Yaskawa INFORM job: SKRZYNIA_5040_90_STOPNI_10BR_OLD.JBI

/JOB
//NAME SKRZYNIA_5040_90_STOPNI_10BR_OLD
//POS
///NPOS 659,659,0,49,0,0
///TOOL 0
///POSTYPE PULSE
///PULSE
C00000=0,-52280,40443,0,6876,0
C00001=82314,-24956,17040,59626,-27382,6248
C00002=93910,-8625,17040,59626,-43355,6248
C00003=98846,-1061,-42166,80308,-57081,-16120
C00004=100452,6057,-48127,85711,-56704,-21322
C00005=96349,29000,-36127,85072,-63022,-26262
C00006=95580,33075,-33256,84644,-64024,-26851
C00007=94197,33846,-32020,85210,-63413,-26698
C00008=95580,33075,-33256,84644,-64024,-26851
C00009=94888,31114,-36362,85298,-63687,-27185
C00010=95580,33075,-33256,84644,-64024,-26851
C00011=95263,33142,-33256,84677,-63995,-26850
C00012=94634,33491,-32695,84935,-63717,-26781
C00013=94130,33776,-32235,85140,-63494,-26725
C00014=95104,32689,-33981,84829,-63917,-26928
C00015=94679,31503,-35865,85229,-63711,-27129
C00016=95263,33142,-33256,84677,-63995,-26850
C00017=95260,33144,-33256,84678,-63995,-26850
C00018=94650,33483,-32714,84929,-63727,-26783
C00019=94112,33789,-32223,85148,-63489,-26723
C00020=95084,32644,-34054,84845,-63909,-26937
C00021=94657,31449,-35950,85247,-63703,-27139
C00022=95260,33144,-33256,84678,-63995,-26850
C00023=95258,33145,-33257,84676,-63996,-26846
C00024=94953,33314,-32988,84801,-63862,-26812
C00025=94037,33833,-32158,85174,-63457,-26709
C00026=94978,32352,-34521,84941,-63860,-26983
C00027=94597,31295,-36193,85297,-63678,-27162
C00028=95258,33145,-33257,84676,-63996,-26846
C00029=95258,33145,-33257,84676,-63996,-26846
C00030=94635,33491,-32703,84932,-63720,-26777
C00031=94255,33706,-32357,85087,-63552,-26734
C00032=95076,32627,-34084,84849,-63906,-26937
C00033=94616,31344,-36119,85281,-63684,-27155
C00034=95258,33145,-33257,84676,-63996,-26846
C00035=95258,25631,32269,66559,-75499,-2416
C00036=95045,25799,32513,66531,-75379,-2372
C00037=94321,26382,33365,66429,-74973,-2219
C00038=95048,24784,31042,66584,-75290,-2483
C00039=94601,23046,28557,66633,-74859,-2609
C00040=95258,25631,32269,66559,-75499,-2416
C00041=98646,19496,-17631,99827,-80462,-21224
C00042=98317,21326,-15127,99395,-81089,-20992
C00043=97962,21529,-14845,99504,-80870,-20995
C00044=98567,20146,-16748,99341,-81286,-21080
C00045=98203,18829,-18537,99489,-81121,-21211
C00046=98811,21047,-15512,99242,-81394,-20987
C00047=98811,19937,1242,97498,-78933,-15296
C00048=98811,19937,1242,97498,-78933,-15296
C00049=98014,20416,1894,97635,-78400,-15298
C00050=98593,19084,88,97564,-78819,-15379
C00051=98194,17557,-1953,97683,-78607,-15521
C00052=98811,19937,1242,97498,-78933,-15296
C00053=98765,34858,63506,90961,-74847,-417
C00054=98962,39103,70654,91062,-76265,452
C00055=98093,40155,72476,90768,-75677,655
C00056=98962,39103,70654,91062,-76265,452
C00057=98539,36034,65455,91246,-76081,-158
C00058=98962,39103,70654,91062,-76265,452
C00059=98994,31803,58419,90917,-73461,-1055
C00060=94428,854,16076,89248,-50738,-4740
C00061=88080,-20128,-3199,80943,-31244,-2335
C00062=48287,-44591,-17414,16172,-14532,25809
C00063=48287,-44591,-17414,16172,-14532,25809
C00064=85348,-13130,13838,41209,-47455,8220
C00065=99199,18818,35660,68259,-73735,-6208
C00066=95720,15423,18785,70454,-68603,-10022
C00067=95720,15423,18785,70454,-68603,-10022
C00068=97055,28839,36684,71776,-79389,-10554
C00069=95990,29701,37981,71658,-78759,-10350
C00070=97055,28839,36684,71776,-79389,-10554
C00071=96570,26656,33448,71832,-78908,-10775
C00072=97055,28839,36684,71776,-79389,-10554
C00073=97055,28839,36684,71776,-79389,-10554
C00074=97055,28839,36684,71776,-79389,-10554
C00075=96028,29668,37934,71662,-78782,-10355
C00076=97055,28839,36684,71776,-79389,-10554
C00077=96569,26658,33449,71833,-78910,-10776
C00078=97055,28839,36684,71776,-79389,-10554
C00079=97055,28839,36684,71776,-79389,-10554
C00080=97055,28839,36684,71776,-79389,-10554
C00081=96073,29634,37879,71669,-78808,-10363
C00082=97055,28839,36684,71776,-79389,-10554
C00083=96556,26588,33346,71835,-78895,-10784
C00084=97055,28839,36684,71776,-79389,-10554
C00085=97055,28839,36684,71776,-79389,-10554
C00086=97055,28839,36684,71776,-79389,-10554
C00087=96070,29634,37881,71667,-78806,-10365
C00088=97055,28839,36684,71776,-79389,-10554
C00089=96542,26531,33264,71837,-78884,-10788
C00090=97055,28839,36684,71776,-79389,-10554
C00091=99222,23346,17795,82202,-78388,4176
C00092=99222,23346,17795,82202,-78388,4176
C00093=98198,24012,18735,82231,-77709,4276
C00094=99222,23346,17795,82202,-78388,4176
C00095=98846,21740,15549,82282,-78105,4028
C00096=99222,23346,17795,82202,-78388,4176
C00097=97305,19304,15511,100837,-75687,4760
C00098=97826,25373,24000,100195,-79238,5786
C00099=96887,26043,24967,100223,-78578,5793
C00100=97826,25373,24000,100195,-79238,5786
C00101=97448,23764,21701,100276,-79072,5588
C00102=97826,25373,24000,100195,-79238,5786
C00103=97826,25373,24000,100195,-79238,5786
C00104=97826,25373,24000,100195,-79238,5786
C00105=96843,26076,25015,100223,-78545,5791
C00106=97826,25373,24000,100195,-79238,5786
C00107=97441,23730,21652,100278,-79068,5583
C00108=97826,25373,24000,100195,-79238,5786
C00109=100071,8792,-2363,102947,-71408,2025
C00110=90699,-12620,-30080,113827,-52438,-6201
C00111=97832,-16290,-36993,112551,-57584,-6005
C00112=83036,-26396,-56580,138157,-49269,-16960
C00113=83036,-26453,-52828,136768,-47205,-15962
C00114=60067,-65836,-77869,147206,-28305,-20439
C00115=63330,-26972,24478,18707,-56801,31483
C00116=95462,-32664,-40336,69376,-39980,4046
C00117=100465,-3562,-10252,69901,-61773,-201
C00118=99635,18997,3540,80919,-74698,-6325
C00119=98097,22561,8426,80415,-76730,-6116
C00120=98097,22561,8426,80415,-76730,-6116
C00121=97377,23028,9077,80478,-76265,-6042
C00122=98097,22561,8426,80415,-76730,-6116
C00123=97807,21406,6827,80497,-76510,-6215
C00124=98097,22561,8426,80415,-76730,-6116
C00125=98899,30801,44624,87834,-79065,838
C00126=98899,30801,44624,87834,-79065,838
C00127=98247,31325,45433,87747,-78622,912
C00128=98899,30801,44624,87834,-79065,838
C00129=98602,29264,42279,87883,-78869,621
C00130=98899,30801,44624,87834,-79065,838
C00131=97973,11446,12587,89117,-68519,-2848
C00132=79911,-29338,-29911,88184,-26074,-2635
C00133=44299,-53382,-38573,-8929,-12050,42418
C00134=44299,-51091,-32799,-7549,-14278,41753
C00135=42754,-66126,12236,-1301,3231,7194
C00136=0,-52280,40443,0,6876,0
C00137=0,-52280,40443,0,6876,0
C00138=0,-43112,23163,-32261,-40956,-29092
C00139=48283,-21883,28214,25170,-26491,-48363
C00140=46664,-3144,58041,18842,-32105,-45325
C00141=50347,-18571,12268,49104,-16423,-60029
C00142=51149,-18702,10839,52647,-16284,-61663
C00143=49023,-16654,12458,50505,-14948,-60880
C00144=50458,-16314,12735,52976,-15639,-61913
C00145=50509,-19000,10610,51503,-15997,-61182
C00146=50509,-19000,10610,51503,-15997,-61182
C00147=51153,-18191,11234,52953,-16222,-61812
C00148=49506,-16603,12499,51322,-15186,-61219
C00149=50699,-16390,12671,53298,-15774,-62041
C00150=50704,-18403,11069,52157,-16018,-61478
C00151=50704,-18403,11069,52157,-16018,-61478
C00152=51011,-18259,11181,52703,-16157,-61707
C00153=49372,-16676,12437,51065,-15128,-61110
C00154=50855,-16321,12727,53567,-15849,-62152
C00155=50704,-18403,11069,52157,-16018,-61478
C00156=50704,-18403,11069,52157,-16018,-61478
C00157=51194,-17966,11787,52443,-16367,-61556
C00158=49641,-16469,12982,50879,-15396,-60984
C00159=51159,-16110,13274,53409,-16135,-62034
C00160=51194,-19029,8982,55593,-15729,-63095
C00161=51005,-17995,11387,52847,-16122,-61778
C00162=51030,-17982,11395,52891,-16135,-61798
C00163=49666,-16664,12446,51542,-15278,-61306
C00164=51234,-16283,12753,54139,-16047,-62382
C00165=51030,-17982,11395,52891,-16135,-61798
C00166=51030,-17982,11395,52891,-16135,-61798
C00167=51056,-17951,11420,52949,-16145,-61823
C00168=49507,-16445,12622,51407,-15172,-61259
C00169=51212,-15994,12989,54262,-16005,-62444
C00170=51056,-17951,11420,52949,-16145,-61823
C00171=50945,-18019,11363,52741,-16103,-61737
C00172=51451,-18380,9957,55416,-15976,-62984
C00173=49638,-16617,11364,53777,-14815,-62399
C00174=51249,-16205,11700,56405,-15635,-63491
C00175=50945,-18019,11363,52741,-16103,-61737
C00176=50945,-18019,11363,52741,-16103,-61737
C00177=51751,-18888,8325,57986,-15754,-64205
C00178=49901,-17096,9744,56519,-14545,-63700
C00179=51443,-16713,10055,58931,-15359,-64698
C00180=50945,-18019,11363,52741,-16103,-61737
C00181=50945,-18019,11363,52741,-16103,-61737
C00182=51752,-17629,11670,54137,-16475,-62321
C00183=49778,-15710,13222,52239,-15234,-61634
C00184=51536,-15216,13634,55124,-16102,-62830
C00185=50945,-18019,11363,52741,-16103,-61737
C00186=50028,-22953,-3957,22347,-31919,-54220
C00187=50556,-22259,-3444,23037,-31901,-54554
C00188=48685,-20311,-1961,21193,-31011,-53711
C00189=50316,-19877,-1623,23110,-31344,-54618
C00190=49456,-22793,-3840,21729,-31736,-53932
C00191=49763,-25421,-36239,24565,-26935,-60445
C00192=49763,-25421,-36239,24565,-26935,-60445
C00193=47682,-22631,-34091,22709,-25786,-59390
C00194=49411,-21994,-33587,24802,-26153,-60557
C00195=49763,-25421,-36239,24565,-26935,-60445
C00196=50713,-12366,-58367,41124,-17813,-74400
C00197=50531,-11018,-57111,41258,-17631,-74434
C00198=49339,-9106,-55286,40470,-17030,-73839
C00199=50327,-8799,-54988,41498,-17395,-74518
C00200=50078,-11370,-57441,40744,-17481,-74102
C00201=49763,-25421,-36239,24565,-26935,-60445
C00202=49426,-25689,-5908,21254,-32432,-53672
C00203=45389,-28224,4312,35967,-15579,-54278
C00204=40154,-51179,-915,24203,-8234,-36524
C00205=0,-52280,40443,0,6876,0
C00206=0,-52280,40443,0,6876,0
C00207=2117,-50103,-33543,4117,45077,-85249
C00208=-26439,-48928,-33543,4117,-52362,-85249
C00209=-26439,-27355,-33543,41485,-52362,-85249
C00210=-47486,-18593,-22655,32887,-41344,-78763
C00211=-48804,2873,-12100,24189,-42468,-81113
C00212=-46457,7101,-11330,26648,-40775,-82885
C00213=-47278,8641,-9483,26175,-40625,-82510
C00214=-46717,9819,-8044,26408,-40882,-82710
C00215=-47278,8641,-9483,26175,-40625,-82510
C00216=-48464,9694,-8203,25521,-40353,-81986
C00217=-47278,8641,-9483,26175,-40625,-82510
C00218=-44522,-635,-31983,49264,-28311,-89687
C00219=-44904,-149,-31453,49090,-28120,-89538
C00220=-44398,873,-30329,49324,-28371,-89731
C00221=-44904,-149,-31453,49090,-28120,-89538
C00222=-45751,485,-30759,48680,-27706,-89207
C00223=-44904,-149,-31453,49090,-28120,-89538
C00224=-41365,-13075,-22481,51159,-38446,-84131
C00225=-20796,-2039,-9686,94158,-57077,-89438
C00226=-24380,-971,-8542,94589,-54660,-89617
C00227=-25651,-542,-8077,94748,-53804,-89683
C00228=-25378,473,-6965,94714,-53986,-89667
C00229=-25651,-542,-8077,94748,-53804,-89683
C00230=-26467,-222,-7729,94854,-53254,-89725
C00231=-25651,-542,-8077,94748,-53804,-89683
C00232=-25651,-542,-8077,94748,-53804,-89683
C00233=-25946,-428,-7954,94785,-53605,-89698
C00234=-25690,517,-6922,94753,-53778,-89686
C00235=-25946,-428,-7954,94785,-53605,-89698
C00236=-26504,-206,-7715,94856,-53230,-89728
C00237=-25946,-428,-7954,94785,-53605,-89698
C00238=-4522,-31762,-35329,90790,-67707,-86470
C00239=34878,-25684,-31064,90205,-94657,-86497
C00240=34878,-25684,-31064,90205,-94657,-86497
C00241=-29329,5838,20653,63819,-53216,-67184
C00242=-29329,5838,20653,63819,-53216,-67184
C00243=-29048,6776,21767,63865,-53412,-67197
C00244=-29329,5838,20653,63819,-53216,-67184
C00245=-29728,6023,20871,63686,-52977,-67114
C00246=-29329,5838,20653,63819,-53216,-67184
C00247=-26603,-1578,11750,66889,-51946,-68995
C00248=-28084,-8635,-16421,94802,-52116,-89609
C00249=-26816,-2974,-10680,94869,-53013,-89721
C00250=-26345,-658,-8205,94838,-53336,-89719
C00251=-26015,535,-6901,94796,-53558,-89702
C00252=-26345,-658,-8205,94838,-53336,-89719
C00253=-26668,-531,-8065,94879,-53120,-89737
C00254=-26345,-658,-8205,94838,-53336,-89719
C00255=-25886,-767,-8323,94779,-53646,-89696
C00256=-25886,-767,-8323,94779,-53646,-89696
C00257=-25568,389,-7061,94741,-53858,-89681
C00258=-25886,-767,-8323,94779,-53646,-89696
C00259=-26674,-459,-7988,94881,-53115,-89738
C00260=-25886,-767,-8323,94779,-53646,-89696
C00261=-25886,-767,-8323,94779,-53646,-89696
C00262=-26039,-1319,-8919,94795,-53542,-89701
C00263=-25594,308,-7149,94744,-53844,-89683
C00264=-26039,-1319,-8919,94795,-53542,-89701
C00265=-26964,-954,-8527,94912,-52922,-89753
C00266=-26039,-1319,-8919,94795,-53542,-89701
C00267=-6422,-16748,-12987,81781,-66398,-84181
C00268=26295,-11282,7080,74868,-91255,-82094
C00269=26295,-11282,7080,74868,-91255,-82094
C00270=-19602,460,18931,65728,-61929,-78089
C00271=-27549,8936,28821,63115,-57256,-76757
C00272=-27549,8936,28821,63115,-57256,-76757
C00273=-27137,10499,30762,63159,-57570,-76739
C00274=-27549,8936,28821,63115,-57256,-76757
C00275=-28395,9323,29301,62815,-56766,-76608
C00276=-27549,8936,28821,63115,-57256,-76757
C00277=-26000,11892,38571,70638,-56518,-75722
C00278=-26000,11892,38571,70638,-56518,-75722
C00279=-25623,13478,40636,70627,-56817,-75642
C00280=-26000,11892,38571,70638,-56518,-75722
C00281=-26799,12251,39037,70343,-56037,-75609
C00282=-26000,11892,38571,70638,-56518,-75722
C00283=-30664,-6343,-14094,96248,-45630,-90223
C00284=-30664,-6343,-14094,96248,-45630,-90223
C00285=-30266,-5205,-12941,96241,-45907,-90235
C00286=-30664,-6343,-14094,96248,-45630,-90223
C00287=-31549,-5956,-13703,96412,-45040,-90299
C00288=-30664,-6343,-14094,96248,-45630,-90223
C00289=-30881,-6301,-14053,96286,-45485,-90239
C00290=-30881,-6301,-14053,96286,-45485,-90239
C00291=-30478,-5160,-12894,96278,-45765,-90250
C00292=-30881,-6301,-14053,96286,-45485,-90239
C00293=-31620,-5975,-13722,96425,-44990,-90303
C00294=-30881,-6301,-14053,96286,-45485,-90239
C00295=-30881,-6301,-14053,96286,-45485,-90239
C00296=-30881,-6301,-14053,96286,-45485,-90239
C00297=-30447,-5069,-12799,96277,-45787,-90250
C00298=-30881,-6301,-14053,96286,-45485,-90239
C00299=-31687,-5947,-13694,96439,-44946,-90310
C00300=-30881,-6301,-14053,96286,-45485,-90239
C00301=-40108,-3695,2740,114838,-35048,-86380
C00302=-40108,-3695,2740,114838,-35048,-86380
C00303=-39569,-2580,3911,114673,-35386,-86267
C00304=-40108,-3695,2740,114838,-35048,-86380
C00305=-40792,-3300,3152,115124,-34647,-86568
C00306=-40108,-3695,2740,114838,-35048,-86380
C00307=-30881,-6301,-14053,96286,-45485,-90239
C00308=-26558,-19284,-27675,95285,-48332,-89713
C00309=-5136,-57382,-50746,80999,-31115,-81799
C00310=-5136,-57382,-50746,80999,-31115,-81799
C00311=-28081,-5880,-3448,89665,-51503,-85625
C00312=-29146,-693,14124,66641,-54461,-78263
C00313=-27186,7805,23879,67003,-55804,-78365
C00314=-27186,7805,23879,67003,-55804,-78365
C00315=-26901,8878,25190,67028,-56018,-78354
C00316=-27186,7805,23879,67003,-55804,-78365
C00317=-27820,8088,24221,66810,-55415,-78267
C00318=-27186,7805,23879,67003,-55804,-78365
C00319=-29983,12431,36540,97303,-47015,-80901
C00320=-29983,5395,14068,105725,-49606,-86937
C00321=-29614,6622,15514,105627,-49820,-86846
C00322=-29983,5395,14068,105725,-49606,-86937
C00323=-30655,5720,14449,105789,-49168,-87017
C00324=-29983,5395,14068,105725,-49606,-86937
C00325=-23275,-722,28392,94611,-50650,-77911
C00326=-23487,-14810,34938,67734,-39470,-58782
C00327=1657,-52280,40443,-304,6876,209
C00328=80083,-25473,16734,55938,-25627,7512
C00329=92674,-9533,16184,58080,-41894,6874
C00330=98391,-2369,-43566,80825,-55961,-16033
C00331=100022,4785,-49618,86526,-55706,-21348
C00332=95373,33537,-36121,86560,-63232,-28029
C00333=93881,36038,-32437,85059,-64562,-27761
C00334=93867,33044,-30650,83528,-64743,-25992
C00335=94930,31411,-33227,84334,-64171,-26252
C00336=94930,31411,-33227,84334,-64171,-26252
C00337=93474,31409,-33627,85103,-63552,-26381
C00338=93474,31409,-33627,85103,-63552,-26381
C00339=96539,31728,-33125,83558,-64961,-26367
C00340=95609,19235,-3385,72159,-68881,-11456
C00341=93675,20756,-1492,72153,-69304,-11461
C00342=93706,20835,-1296,72059,-69329,-11411
C00343=95041,22056,296,71883,-70234,-11460
C00344=95041,22056,296,71883,-70234,-11460
C00345=93716,20674,-1606,72153,-69328,-11471
C00346=93749,20787,-1450,72141,-69355,-11463
C00347=95041,22056,296,71883,-70234,-11460
C00348=95041,22056,296,71883,-70234,-11460
C00349=93853,20645,-1646,72134,-69414,-11487
C00350=93701,20690,-1585,72152,-69318,-11471
C00351=95606,21673,-233,71830,-70568,-11545
C00352=95936,-8790,-36169,76308,-52611,-10237
C00353=87381,-35372,-46042,66676,-50803,-1891
C00354=84950,-62287,8062,38288,-37295,1216
C00355=1657,-52280,40443,-304,6876,209
C00356=1657,-52280,40443,-304,6876,209
C00357=841,-50033,-33518,5341,45264,-86395
C00358=-28809,-48989,-33566,1638,-52261,-83793
C00359=-27557,-28108,-34083,40495,-51335,-84423
C00360=-40439,-25215,-42205,50808,-38049,-86084
C00361=-38463,-7029,-29048,56299,-36479,-89524
C00362=-47795,3485,-15813,29932,-36086,-79941
C00363=-43904,4858,-16350,36941,-37959,-85674
C00364=828,-25363,-17205,45133,-71673,-88219
C00365=4678,-17958,4683,47898,-79597,-85332
C00366=-18355,-35625,17567,22328,-38004,-35198
C00367=38277,-55351,-7622,112862,-31065,-32489
C00368=1657,-52280,40443,-304,6876,209
C00369=-4811,-36310,24637,-49210,-33845,-31988
C00370=41748,-30202,7105,17690,-22932,-42913
C00371=41748,-30202,7105,17690,-22932,-42913
C00372=49037,-21406,10886,33705,-21312,-49933
C00373=57938,-18196,5914,66765,-23183,-68504
C00374=62071,-18819,1330,80566,-26873,-76175
C00375=48249,-23742,8050,33819,-21114,-50004
C00376=-4811,-36310,24637,-49210,-33845,-31988
C00377=1657,-52280,40443,-304,6876,209
C00378=1613,-52280,40443,-296,6876,203
C00379=73560,-62084,7826,28695,-34737,3666
C00380=88377,-34186,-45291,67238,-52212,-2442
C00381=96528,-7533,-34932,76119,-53878,-10439
C00382=100432,21324,12575,83706,-77956,-7498
C00383=98573,22459,14150,83808,-76714,-7352
C00384=97684,25950,19098,83414,-79070,-7056
C00385=97598,25982,19143,83418,-79013,-7051
C00386=99338,18438,8643,84272,-74238,-7648
C00387=99336,18440,8642,84276,-74234,-7647
C00388=97786,25707,18749,83415,-79135,-7087
C00389=97740,25808,18892,83414,-79103,-7073
C00390=99336,18440,8642,84276,-74234,-7647
C00391=99336,18440,8642,84276,-74234,-7647
C00392=97857,25790,18866,83408,-79181,-7079
C00393=97666,25767,18833,83421,-79056,-7078
C00394=99336,18440,8642,84276,-74234,-7647
C00395=100441,9433,14994,80938,-68243,-1963
C00396=98851,2841,7216,80537,-62817,-1838
C00397=99868,-33,22146,72719,-59601,5126
C00398=99028,-10516,17309,71061,-60695,4227
C00399=58820,-39124,10926,53325,-41870,3759
C00400=0,-52280,40443,0,6876,0
C00401=37281,-50778,-9546,79570,-75313,-71156
C00402=21038,-23698,-30323,82948,-81132,-85647
C00403=7436,-16003,-3781,101119,-69483,-78457
C00404=-27121,-5377,5501,98364,-47418,-81834
C00405=-29080,8413,23722,96931,-48705,-80906
C00406=-31669,8189,15332,113614,-50161,-86745
C00407=-29309,2640,17780,96201,-45535,-80500
C00408=-23641,-6994,7554,96186,-49257,-79992
C00409=19501,-22886,-23351,116550,-78011,-79854
C00410=32334,-18287,-16541,87042,-89296,-82607
C00411=-25600,-16732,-29668,75447,-47301,-83964
C00412=-31045,-6665,-14727,69712,-44450,-80944
C00413=-32809,-4927,-18520,77308,-42173,-84100
C00414=-33573,-4913,-21143,75716,-41103,-84515
C00415=-32065,-7067,-21213,73988,-42430,-83589
C00416=-38755,-17773,-33721,67311,-34017,-81961
C00417=-35581,-11023,-27644,69090,-35721,-83210
C00418=-30590,527,-16574,72341,-46994,-87004
C00419=-30590,212,-22171,75529,-46132,-89216
C00420=-33949,-22068,-37275,67306,-37324,-82274
C00421=-40042,-68802,-18337,47708,-19461,-45384
C00422=-37287,-55159,35520,2191,5667,-2084
C00423=0,-52280,40443,0,6876,0
C00424=0,-36700,24612,-42871,-31823,-33862
C00425=44403,-30110,7154,24155,-23805,-45557
C00426=48366,-23967,9999,33441,-23050,-49710
C00427=57059,-21871,4355,62840,-24072,-66406
C00428=62704,-18615,1157,81482,-27976,-78161
C00429=66087,-18332,-2621,91395,-32291,-83757
C00430=50677,-23266,8367,38735,-22212,-52049
C00431=47073,-34549,9488,27883,-30316,-51458
C00432=0,-52280,40443,0,6876,0
C00433=0,-52280,40443,0,6876,0
C00434=73560,-62084,7826,28695,-34737,3666
C00435=87376,-41373,-10333,58133,-51016,401
C00436=100341,-12426,-15111,78591,-60044,-5220
C00437=100467,-7393,-15195,81625,-60158,-6002
C00438=99336,18440,8642,84276,-74234,-7647
C00439=98831,26826,38209,85264,-77545,-1440
C00440=97968,30695,40017,90402,-79732,-2682
C00441=98020,30578,39840,90409,-79769,-2698
C00442=101143,13060,5845,92851,-72534,-7825
C00443=98403,-20338,-58596,109487,-56658,-19777
C00444=60204,-59872,-73451,117647,-17639,-18840
C00445=73315,-17786,32032,37482,-51892,27783
C00446=73315,-17786,32032,37482,-51892,27783
C00447=95648,9329,59164,52594,-59741,22349
C00448=95648,-19617,-26605,79265,-44876,2231
C00449=83785,-15028,-22673,79363,-36769,2523
C00450=91376,-7063,-15168,80845,-51819,703
C00451=99322,22762,20659,79494,-77572,134
C00452=99123,22953,21148,79461,-77463,232
C00453=98877,27968,32487,76173,-79945,2468
C00454=95369,26181,23160,71095,-76769,901
C00455=95369,28262,32501,70203,-78207,3099
C00456=100802,24456,20984,80151,-80320,-697
C00457=99662,22785,17568,82066,-77607,-1267
C00458=97757,25456,21360,81884,-78797,-1037
C00459=97789,25433,21327,81884,-78819,-1041
C00460=99676,21999,16470,82145,-76972,-1318
C00461=97441,-6012,-18634,86114,-58345,-2339
C00462=92377,-33385,-41303,83059,-36844,1354
C00463=79425,-37128,-15462,51820,-35721,18807
C00464=43180,-50572,-20637,6552,-29302,38834
C00465=37721,-67612,11381,1325,-438,7850
C00466=-37287,-55159,35520,2191,5667,-2084
C00467=-40042,-68802,-18337,47708,-19461,-45384
C00468=-28646,-23138,-32952,89786,-42552,-85395
C00469=-30193,-12825,-24186,91372,-43752,-86505
C00470=-31120,-5451,-17038,91814,-44683,-86873
C00471=-31134,-5488,-17074,91814,-44673,-86872
C00472=-30706,-9539,-21090,91641,-44141,-86712
C00473=-30706,-9539,-21090,91641,-44141,-86712
C00474=-33095,-7143,-18859,92591,-41579,-87147
C00475=-33112,-7185,-18903,92591,-41567,-87145
C00476=-33746,-1176,10845,101603,-40605,-81585
C00477=-10974,-25157,-10641,98520,-54806,-77487
C00478=31369,-21210,-7704,102203,-82608,-74705
C00479=31369,-21210,-7704,102203,-82608,-74705
C00480=32236,-17736,2151,73206,-90006,-78496
C00481=2413,-16607,2080,65101,-71431,-76259
C00482=-34840,2394,22974,48249,-51640,-69452
C00483=-33831,18589,49739,44880,-63097,-61844
C00484=-33831,13710,36104,47061,-59222,-64049
C00485=-35408,1628,18221,49605,-49628,-70543
C00486=-36029,-1090,16876,49320,-48191,-69422
C00487=-45963,-23918,13188,27154,-34733,-49172
C00488=0,-52280,40443,0,6876,0
C00489=37164,-60659,6466,13301,-5027,-19773
C00490=45362,-39990,2831,27538,-17767,-40935
C00491=55315,-20486,12421,43917,-25084,-54085
C00492=61760,-17076,4399,78300,-26495,-75523
C00493=66887,-15221,5723,82563,-32969,-76938
C00494=53534,-30170,6270,37667,-26637,-51098
C00495=41180,-61187,4729,17280,-8498,-23442
C00496=0,-52280,40443,0,6876,0
C00497=0,-52280,40443,0,6876,0
C00498=37721,-67612,11381,1325,-438,7850
C00499=43180,-50572,-20637,6552,-29302,38834
C00500=79425,-37128,-15462,51820,-35721,18807
C00501=92377,-33385,-41303,83059,-36844,1354
C00502=100252,-4949,-17551,85890,-60241,-2391
C00503=99662,22785,17568,82066,-77607,-1267
C00504=98003,26711,23176,81782,-79695,-932
C00505=98187,26766,23256,81772,-79821,-932
C00506=99662,22785,17568,82066,-77607,-1267
C00507=99662,22785,17568,82066,-77607,-1267
C00508=97671,26258,22515,81825,-79282,-965
C00509=97727,26283,22551,81822,-79321,-966
C00510=99662,22785,17568,82066,-77607,-1267
C00511=99662,22785,17568,82066,-77607,-1267
C00512=97804,25700,21708,81856,-79094,-1026
C00513=97599,25610,21578,81868,-78954,-1030
C00514=99662,22785,17568,82066,-77607,-1267
C00515=97206,-2526,-13508,84298,-60212,-1778
C00516=99581,-17537,-27968,84120,-53285,-833
C00517=87335,-30812,-23405,71152,-48070,8074
C00518=43180,-50572,-20637,6552,-29302,38834
C00519=37721,-67612,11381,1325,-438,7850
C00520=0,-52280,40443,0,6876,0
C00521=0,-52280,40443,0,6876,0
C00522=-37287,-55159,35520,2191,5667,-2084
C00523=-40042,-68802,-18337,47708,-19461,-45384
C00524=-46318,-50945,-29177,106898,-20771,-78142
C00525=-46775,-41793,-28600,116864,-25974,-84568
C00526=-37035,-31234,-22655,117900,-33576,-84505
C00527=-33623,-10331,-13330,109256,-42555,-87094
C00528=-33459,-4510,-9104,107028,-43857,-87640
C00529=-36854,1758,5452,119173,-43239,-89918
C00530=-43373,7690,30281,135695,-33936,-89271
C00531=-40042,-68802,-18337,47708,-19461,-45384
C00532=-37287,-55159,35520,2191,5667,-2084
C00533=0,-52280,40443,0,6876,0
C00534=0,-52280,40443,0,-40770,0
C00535=-67457,-24715,25918,-9670,-26808,-27227
C00536=-30973,4607,39277,65194,-48165,-66059
C00537=-30973,4607,39277,65194,-48165,-66059
C00538=-26559,20289,58443,71098,-56573,-67847
C00539=-26559,30445,82576,66093,-59546,-63271
C00540=-30973,4607,39277,65194,-48165,-66059
C00541=-30973,4607,39277,65194,-48165,-66059
C00542=-27009,20890,60963,69173,-56615,-66199
C00543=-27009,34969,93454,62905,-61033,-60343
C00544=-30973,4607,39277,65194,-48165,-66059
C00545=-35251,-18143,20376,53513,-41117,-59413
C00546=-9534,-43450,13514,26959,-29486,-38723
C00547=-22834,-59963,22946,6692,-2150,-9612
C00548=0,-52280,40443,0,6876,0
C00549=23708,-46776,23536,16027,-4787,-19738
C00550=50917,-40459,4132,34421,-18173,-42391
C00551=55315,-20486,12421,43917,-25084,-54085
C00552=52021,-27344,-11614,25442,-32756,-51822
C00553=62388,-19076,-7315,47741,-37100,-57915
C00554=60492,-23043,-43968,60514,-28343,-68592
C00555=52021,-27344,-11614,25442,-32756,-51822
C00556=46096,-45842,-2681,20981,-19497,-36310
C00557=41180,-61187,4729,17280,-8498,-23442
C00558=0,-52280,40443,0,6876,0
C00559=0,-52280,40443,0,6876,0
C00560=37721,-67612,11381,1325,-438,7850
C00561=43180,-50572,-20637,6552,-29302,38834
C00562=79425,-37128,-15462,51820,-35721,18807
C00563=92377,-33385,-41303,83059,-36844,1354
C00564=97441,-6012,-18634,86114,-58345,-2339
C00565=98203,16433,5975,106740,-76906,-7461
C00566=95380,23681,15858,105888,-79485,-6352
C00567=95372,23687,15868,105888,-79480,-6352
C00568=95494,24167,16550,105816,-79738,-6257
C00569=95392,24052,16387,105831,-79681,-6279
C00570=95324,24045,16377,105840,-79638,-6287
C00571=98203,16433,5975,106740,-76906,-7461
C00572=100438,3826,-9542,108367,-72171,-8932
C00573=98957,-20219,-27813,100777,-56896,-5666
C00574=87335,-30812,-23405,71152,-48070,8074
C00575=80632,-38079,-20908,64053,-45216,12949
C00576=43180,-50572,-20637,6552,-29302,38834
C00577=37721,-67612,11381,1325,-438,7850
C00578=0,-52280,40443,0,6876,0
C00579=-54026,-30203,28811,-7745,-28969,-5087
C00580=-81492,-18979,22896,-11682,-23662,-26316
C00581=-31639,1998,34377,78496,-41866,-64115
C00582=-28167,19375,56310,81342,-50085,-63750
C00583=-28167,28622,78575,74894,-51467,-58871
C00584=-33078,8378,41935,77523,-41039,-63739
C00585=-46905,3098,9726,144001,-39915,-89043
C00586=-37647,13740,22660,131317,-50520,-79512
C00587=-37647,16845,33202,128344,-47106,-77354
C00588=-46905,3098,9726,144001,-39915,-89043
C00589=-42864,18028,43807,131618,-37529,-87119
C00590=-44052,21146,48203,131480,-36504,-87179
C00591=-44605,22126,50160,132440,-35973,-87409
C00592=-42864,18028,43807,131618,-37529,-87119
C00593=-32723,6704,21658,111173,-45396,-82543
C00594=-34422,-9999,20796,72411,-42519,-66994
C00595=-35251,-18143,20376,53513,-41117,-59413
C00596=-9534,-43450,13514,26959,-29486,-38723
C00597=-22834,-59963,22946,6692,-2150,-9612
C00598=0,-52280,40443,0,6876,0
C00599=23708,-46776,23536,16027,-4787,-19738
C00600=50917,-40459,4132,34421,-18173,-42391
C00601=56351,-28617,-8977,50177,-24220,-59041
C00602=56351,-28617,-8977,50177,-24220,-59041
C00603=61013,-25727,-20437,91852,-25479,-87385
C00604=68741,-23000,-19911,95900,-36007,-87783
C00605=59870,-32730,-20784,77712,-26701,-76039
C00606=36994,-41399,-15582,14937,-21377,-43241
C00607=31287,-69981,-10850,7253,-6843,-20996
C00608=19644,-57271,30737,863,5243,-2499
C00609=0,-52280,40443,0,6876,0
C00610=0,-52280,40443,0,6876,0
C00611=37721,-67612,11381,1325,-438,7850
C00612=43180,-50572,-20637,6552,-29302,38834
C00613=92325,-23846,-7228,63960,-40898,12898
C00614=83562,-2075,23934,52242,-47081,17120
C00615=81926,-4528,18929,54087,-44625,16400
C00616=98156,27605,40467,74304,-79249,6093
C00617=97389,28448,36068,78537,-79231,3814
C00618=97907,24801,21502,85617,-78711,-660
C00619=99547,21785,17244,85874,-76675,-945
C00620=99547,21785,17244,85875,-76675,-945
C00621=97758,24649,21282,85635,-78482,-675
C00622=97758,26167,28392,84986,-78619,1092
C00623=99547,21785,17244,85875,-76675,-945
C00624=98541,21134,18604,96699,-76883,-2153
C00625=97093,25194,24413,97463,-78486,-1748
C00626=97108,27415,33780,96610,-77663,471
C00627=100501,23939,19565,97610,-81211,-2656
C00628=99547,21785,17244,85875,-76675,-945
C00629=85644,-16652,-26140,89995,-40279,-1638
C00630=96357,-21723,-30363,88205,-47532,-883
C00631=98913,1421,32623,59426,-59934,14740
C00632=68865,-35989,-5252,49829,-38105,21179
C00633=80632,-38079,-20908,64053,-45216,12949
C00634=43180,-50572,-20637,6552,-29302,38834
C00635=37721,-67612,11381,1325,-438,7850
C00636=0,-52280,40443,0,6876,0
C00637=0,-52278,40443,0,6872,5
C00638=0,-52278,40443,31822,-65283,-46097
C00639=-7673,2330,44178,76838,-66870,-70196
C00640=-24298,4331,21590,82032,-53834,-78397
C00641=-25374,11897,30998,81913,-55707,-77909
C00642=-25374,16253,43677,78456,-56404,-74921
C00643=-24298,4331,21590,82032,-53834,-78397
C00644=3014,-20441,-7349,104591,-68614,-79454
C00645=17388,-18739,-2459,99831,-77693,-75560
C00646=13238,-21720,-1359,93359,-59492,-72612
C00647=-10261,-46634,14475,36899,-22136,-31570
C00648=-22834,-59963,22946,6692,-2150,-9612
C00649=0,-52280,40443,0,6876,0
C00650=23708,-46776,23536,16027,-4787,-19738
C00651=50917,-40459,4132,34421,-18173,-42391
C00652=55315,-20486,12421,43917,-25084,-54085
C00653=52609,-18323,14042,41333,-23544,-53138
C00654=70054,-15959,-1295,94448,-37577,-86566
C00655=61757,-17157,6384,73937,-27308,-72117
C00656=37618,-28118,7425,14704,-21495,-41826
C00657=31287,-69981,-10850,7253,-6843,-20996
C00658=0,-52280,40443,0,6876,0
BC00000=468276
BC00001=445130
BC00002=445130
BC00003=445130
BC00004=445130
BC00005=445130
BC00006=445130
BC00007=445130
BC00008=445130
BC00009=445130
BC00010=445130
BC00011=491232
BC00012=491232
BC00013=491232
BC00014=491232
BC00015=491232
BC00016=491232
BC00017=537442
BC00018=537442
BC00019=537442
BC00020=537442
BC00021=537442
BC00022=537442
BC00023=583546
BC00024=583546
BC00025=583546
BC00026=583546
BC00027=583546
BC00028=583546
BC00029=606594
BC00030=606594
BC00031=606594
BC00032=606594
BC00033=606594
BC00034=606594
BC00035=559393
BC00036=559393
BC00037=559393
BC00038=559393
BC00039=559393
BC00040=559393
BC00041=605503
BC00042=605503
BC00043=605503
BC00044=605503
BC00045=605503
BC00046=605503
BC00047=605503
BC00048=605503
BC00049=605503
BC00050=605503
BC00051=605503
BC00052=605503
BC00053=604255
BC00054=604255
BC00055=604255
BC00056=604255
BC00057=604255
BC00058=604255
BC00059=604255
BC00060=604255
BC00061=604255
BC00062=604255
BC00063=699121
BC00064=714117
BC00065=714117
BC00066=714117
BC00067=714117
BC00068=714117
BC00069=714117
BC00070=714117
BC00071=714117
BC00072=714117
BC00073=737203
BC00074=737203
BC00075=737203
BC00076=737203
BC00077=737203
BC00078=737203
BC00079=783275
BC00080=783275
BC00081=783275
BC00082=783275
BC00083=783275
BC00084=783275
BC00085=806363
BC00086=806363
BC00087=806363
BC00088=806363
BC00089=806363
BC00090=806363
BC00091=843190
BC00092=843190
BC00093=843190
BC00094=843190
BC00095=843190
BC00096=843190
BC00097=849204
BC00098=849204
BC00099=849204
BC00100=849204
BC00101=849204
BC00102=849204
BC00103=872244
BC00104=872244
BC00105=872244
BC00106=872244
BC00107=872244
BC00108=872244
BC00109=872244
BC00110=872244
BC00111=872244
BC00112=872244
BC00113=872244
BC00114=872244
BC00115=914118
BC00116=976590
BC00117=976590
BC00118=976734
BC00119=976734
BC00120=976734
BC00121=976734
BC00122=976734
BC00123=976734
BC00124=976734
BC00125=973058
BC00126=973058
BC00127=973058
BC00128=973058
BC00129=973058
BC00130=973058
BC00131=984446
BC00132=994872
BC00133=996146
BC00134=935999
BC00135=857759
BC00136=811793
BC00137=811793
BC00138=811795
BC00139=919701
BC00140=919701
BC00141=949003
BC00142=951100
BC00143=951100
BC00144=951100
BC00145=951100
BC00146=889624
BC00147=889624
BC00148=889624
BC00149=889624
BC00150=889624
BC00151=828182
BC00152=828182
BC00153=828182
BC00154=828182
BC00155=828182
BC00156=766752
BC00157=766752
BC00158=766752
BC00159=766752
BC00160=766752
BC00161=705350
BC00162=705350
BC00163=705350
BC00164=705350
BC00165=705350
BC00166=647188
BC00167=647188
BC00168=647188
BC00169=647188
BC00170=647188
BC00171=582464
BC00172=582464
BC00173=582464
BC00174=582464
BC00175=582464
BC00176=520992
BC00177=520992
BC00178=520992
BC00179=520992
BC00180=520992
BC00181=459540
BC00182=459540
BC00183=459540
BC00184=459540
BC00185=459540
BC00186=459544
BC00187=459544
BC00188=459544
BC00189=459544
BC00190=459544
BC00191=459544
BC00192=459544
BC00193=459544
BC00194=459544
BC00195=459544
BC00196=459544
BC00197=459544
BC00198=459544
BC00199=459544
BC00200=459544
BC00201=459544
BC00202=459544
BC00203=459540
BC00204=533216
BC00205=533216
BC00206=492150
BC00207=423885
BC00208=423885
BC00209=423885
BC00210=493160
BC00211=493160
BC00212=493160
BC00213=493160
BC00214=493160
BC00215=493160
BC00216=493160
BC00217=493160
BC00218=539180
BC00219=539180
BC00220=539180
BC00221=539180
BC00222=539180
BC00223=539180
BC00224=495049
BC00225=485388
BC00226=485384
BC00227=485384
BC00228=485384
BC00229=485384
BC00230=485384
BC00231=485384
BC00232=508449
BC00233=508449
BC00234=508449
BC00235=508449
BC00236=508449
BC00237=508449
BC00238=485386
BC00239=485386
BC00240=600790
BC00241=562212
BC00242=562212
BC00243=562212
BC00244=562212
BC00245=562212
BC00246=562212
BC00247=563312
BC00248=600589
BC00249=600589
BC00250=600589
BC00251=600589
BC00252=600589
BC00253=600589
BC00254=600589
BC00255=623637
BC00256=623637
BC00257=623637
BC00258=623637
BC00259=623637
BC00260=623637
BC00261=669704
BC00262=669704
BC00263=669704
BC00264=669704
BC00265=669704
BC00266=669704
BC00267=658366
BC00268=643307
BC00269=740888
BC00270=738443
BC00271=715786
BC00272=715786
BC00273=715785
BC00274=715786
BC00275=715786
BC00276=715786
BC00277=715786
BC00278=715786
BC00279=715786
BC00280=715786
BC00281=715786
BC00282=715786
BC00283=784942
BC00284=784942
BC00285=784942
BC00286=784942
BC00287=784942
BC00288=784942
BC00289=807985
BC00290=807985
BC00291=807985
BC00292=807985
BC00293=807985
BC00294=807985
BC00295=854090
BC00296=854090
BC00297=854090
BC00298=854090
BC00299=854090
BC00300=854090
BC00301=854090
BC00302=854090
BC00303=854090
BC00304=854090
BC00305=854090
BC00306=854090
BC00307=854090
BC00308=854090
BC00309=854090
BC00310=990684
BC00311=984461
BC00312=984658
BC00313=984658
BC00314=984658
BC00315=984658
BC00316=984658
BC00317=984658
BC00318=984658
BC00319=969297
BC00320=969297
BC00321=969297
BC00322=969297
BC00323=969297
BC00324=969297
BC00325=940619
BC00326=920377
BC00327=445130
BC00328=445130
BC00329=445130
BC00330=445130
BC00331=445130
BC00332=445130
BC00333=445130
BC00334=445722
BC00335=445722
BC00336=484130
BC00337=492273
BC00338=481757
BC00339=492273
BC00340=473247
BC00341=480983
BC00342=473247
BC00343=480984
BC00344=519335
BC00345=527043
BC00346=519335
BC00347=519335
BC00348=542403
BC00349=550079
BC00350=542403
BC00351=542207
BC00352=542207
BC00353=542207
BC00354=542207
BC00355=542207
BC00356=492150
BC00357=423885
BC00358=423885
BC00359=423885
BC00360=423885
BC00361=423885
BC00362=481098
BC00363=480936
BC00364=454901
BC00365=477799
BC00366=477799
BC00367=477799
BC00368=493160
BC00369=582810
BC00370=655182
BC00371=655182
BC00372=655182
BC00373=655182
BC00374=716642
BC00375=716642
BC00376=582810
BC00377=493160
BC00378=494470
BC00379=542207
BC00380=542207
BC00381=590944
BC00382=543764
BC00383=543764
BC00384=551528
BC00385=543764
BC00386=551454
BC00387=589824
BC00388=597582
BC00389=589882
BC00390=589824
BC00391=612873
BC00392=620666
BC00393=612946
BC00394=612873
BC00395=612873
BC00396=612873
BC00397=584417
BC00398=584417
BC00399=584417
BC00400=584417
BC00401=542360
BC00402=521200
BC00403=436412
BC00404=459757
BC00405=459757
BC00406=459757
BC00407=459757
BC00408=427483
BC00409=427483
BC00410=592276
BC00411=597260
BC00412=598004
BC00413=598004
BC00414=598004
BC00415=598004
BC00416=650931
BC00417=650931
BC00418=658595
BC00419=658595
BC00420=658595
BC00421=620193
BC00422=620193
BC00423=620193
BC00424=812803
BC00425=887783
BC00426=893694
BC00427=897534
BC00428=900962
BC00429=962387
BC00430=962387
BC00431=853059
BC00432=542207
BC00433=542207
BC00434=542207
BC00435=532286
BC00436=583284
BC00437=590944
BC00438=612873
BC00439=625395
BC00440=625395
BC00441=633159
BC00442=633159
BC00443=633159
BC00444=633159
BC00445=633159
BC00446=681733
BC00447=681733
BC00448=740703
BC00449=740703
BC00450=740703
BC00451=740703
BC00452=710007
BC00453=710007
BC00454=721641
BC00455=721641
BC00456=724045
BC00457=727159
BC00458=725395
BC00459=733103
BC00460=733103
BC00461=733103
BC00462=733103
BC00463=733103
BC00464=733103
BC00465=733103
BC00466=620193
BC00467=620193
BC00468=635598
BC00469=635598
BC00470=635598
BC00471=643271
BC00472=641590
BC00473=681683
BC00474=681683
BC00475=689331
BC00476=620239
BC00477=620239
BC00478=620239
BC00479=749060
BC00480=763078
BC00481=749658
BC00482=735414
BC00483=735414
BC00484=735414
BC00485=727742
BC00486=736137
BC00487=709811
BC00488=620193
BC00489=561542
BC00490=498768
BC00491=407896
BC00492=407891
BC00493=469397
BC00494=469397
BC00495=524165
BC00496=524165
BC00497=733103
BC00498=733103
BC00499=733103
BC00500=733103
BC00501=733103
BC00502=733103
BC00503=771424
BC00504=771424
BC00505=779179
BC00506=771424
BC00507=794504
BC00508=794504
BC00509=802184
BC00510=794504
BC00511=840598
BC00512=840598
BC00513=848318
BC00514=840598
BC00515=840598
BC00516=840598
BC00517=840598
BC00518=795297
BC00519=733103
BC00520=733103
BC00521=584417
BC00522=620193
BC00523=620193
BC00524=612942
BC00525=610379
BC00526=610379
BC00527=658993
BC00528=670151
BC00529=646716
BC00530=593346
BC00531=585637
BC00532=620193
BC00533=620193
BC00534=722068
BC00535=722068
BC00536=744765
BC00537=742336
BC00538=742336
BC00539=742336
BC00540=742336
BC00541=765388
BC00542=765388
BC00543=765388
BC00544=765388
BC00545=750104
BC00546=672725
BC00547=672725
BC00548=672725
BC00549=576077
BC00550=465158
BC00551=407896
BC00552=407896
BC00553=407896
BC00554=407896
BC00555=407896
BC00556=471446
BC00557=524165
BC00558=524165
BC00559=733103
BC00560=733103
BC00561=733103
BC00562=733103
BC00563=733103
BC00564=733103
BC00565=846020
BC00566=846020
BC00567=853796
BC00568=869044
BC00569=869044
BC00570=876836
BC00571=869044
BC00572=869044
BC00573=860147
BC00574=840598
BC00575=840598
BC00576=795297
BC00577=733103
BC00578=733103
BC00579=762701
BC00580=791880
BC00581=794999
BC00582=794999
BC00583=794999
BC00584=794999
BC00585=823302
BC00586=823302
BC00587=823302
BC00588=823302
BC00589=823302
BC00590=823302
BC00591=829334
BC00592=823302
BC00593=823302
BC00594=774095
BC00595=750104
BC00596=672725
BC00597=672725
BC00598=672725
BC00599=576077
BC00600=513681
BC00601=557970
BC00602=557970
BC00603=557404
BC00604=618554
BC00605=618492
BC00606=618402
BC00607=618402
BC00608=618402
BC00609=618402
BC00610=733103
BC00611=733103
BC00612=931156
BC00613=923671
BC00614=923671
BC00615=923671
BC00616=947035
BC00617=946859
BC00618=954731
BC00619=954731
BC00620=993094
BC00621=993094
BC00622=994811
BC00623=993094
BC00624=993603
BC00625=993603
BC00626=993603
BC00627=993603
BC00628=993094
BC00629=993094
BC00630=993094
BC00631=954137
BC00632=952322
BC00633=840598
BC00634=795297
BC00635=733103
BC00636=733103
BC00637=834980
BC00638=921533
BC00639=949466
BC00640=969584
BC00641=969584
BC00642=969584
BC00643=969584
BC00644=963295
BC00645=944127
BC00646=908449
BC00647=754884
BC00648=672725
BC00649=672725
BC00650=749842
BC00651=756681
BC00652=776639
BC00653=776639
BC00654=776639
BC00655=837995
BC00656=837995
BC00657=742282
BC00658=742282
///POSTYPE BASE
///RECTAN
///RCONF 1,0,0,0,0,0,0,0,0,0,0,0,0,0,0,0,0,0,0,0,0,0,0,0
P00006=0.000,0.000,0.000,0.0000,0.0000,0.0000
///RCONF 0,0,0,0,0,0,0,0,0,0,0,0,0,0,0,0,0,0,0,0,0,0,0,0
P00058=0.000,0.000,3.000,0.0000,0.0000,0.0000
///RCONF 1,0,0,0,0,0,0,0,0,0,0,0,0,0,0,0,0,0,0,0,0,0,0,0
P00300=-0.036,-1.505,2.318,0.0000,0.0000,0.0000
///RCONF 0,0,0,0,0,0,0,0,0,0,0,0,0,0,0,0,0,0,0,0,0,0,0,0
P00301=0.005,-4.708,-4.628,0.0000,0.0000,0.0000
P00302=0.052,-2.937,-4.426,0.0000,0.0000,0.0000
P00303=-0.004,-1.437,-4.584,0.0000,0.0000,0.0000
P00304=0.028,-1.666,-4.234,0.0000,0.0000,0.0000
P00305=-0.003,-1.920,-3.501,0.0000,0.0000,0.0000
P00306=0.015,-2.252,-3.054,0.0000,0.0000,0.0000
P00307=0.019,-2.151,-5.077,0.0000,0.0000,0.0000
P00308=-0.003,-2.092,-4.888,0.0000,0.0000,0.0000
P00309=-0.040,-2.205,-4.992,0.0000,0.0000,0.0000
P00310=-0.006,-2.490,-5.925,0.0000,0.0000,0.0000
P00311=-0.007,-2.079,-5.307,0.0000,0.0000,0.0000
P00312=-0.032,2.202,-7.632,0.0000,0.0000,0.0000
///RCONF 1,0,0,0,0,0,0,0,0,0,0,0,0,0,0,0,0,0,0,0,0,0,0,0
P00313=-0.088,1.055,2.110,0.0000,0.0000,0.0000
P00314=-0.055,1.752,1.634,0.0000,0.0000,0.0000
P00315=-0.074,0.897,1.645,0.0000,0.0000,0.0000
P00316=0.009,2.112,2.075,0.0000,0.0000,0.0000
P00317=-0.015,2.781,3.126,0.0000,0.0000,0.0000
///RCONF 0,0,0,0,0,0,0,0,0,0,0,0,0,0,0,0,0,0,0,0,0,0,0,0
P00350=11.519,-0.008,1.149,0.0000,0.0000,0.0000
P00351=13.563,-0.027,-0.653,0.0000,0.0000,0.0000
P00352=13.252,-0.027,-0.827,0.0000,0.0000,0.0000
P00353=10.971,-0.082,0.776,0.0000,0.0000,0.0000
P00354=-0.024,2.508,-1.824,0.0000,0.0000,0.0000
P00355=-0.001,2.528,-1.131,0.0000,0.0000,0.0000
P00356=-0.034,2.921,-0.262,0.0000,0.0000,0.0000
P00357=0.003,3.386,-0.091,0.0000,0.0000,0.0000
P00358=0.014,3.037,-0.020,0.0000,0.0000,0.0000
P00359=-0.005,2.731,0.912,0.0000,0.0000,0.0000
P00360=-0.011,3.412,0.438,0.0000,0.0000,0.0000
P00361=0.018,3.050,1.253,0.0000,0.0000,0.0000
P00401=3.430,-0.021,1.131,0.0000,0.0000,0.0000
P00402=-0.253,1.107,3.062,0.0000,0.0000,0.0000
P00403=-3.666,-0.015,5.328,0.0000,0.0000,0.0000
///RCONF 1,0,0,0,0,0,0,0,0,0,0,0,0,0,0,0,0,0,0,0,0,0,0,0
P00404=0.029,4.189,-1.030,0.0000,0.0000,0.0000
///RCONF 0,0,0,0,0,0,0,0,0,0,0,0,0,0,0,0,0,0,0,0,0,0,0,0
P00405=2.420,0.007,1.427,0.0000,0.0000,0.0000
P00406=3.513,-0.022,0.429,0.0000,0.0000,0.0000
///RCONF 1,0,0,0,1,0,0,0,0,0,0,0,0,0,0,0,0,0,0,0,0,0,0,0
P00407=-0.029,2.348,-1.469,0.0000,0.0000,0.0000
P00408=0.010,1.346,-1.479,0.0000,0.0000,0.0000
///RCONF 1,0,0,0,0,0,0,0,0,0,0,0,0,0,0,0,0,0,0,0,0,0,0,0
P00409=-0.026,2.090,-1.483,0.0000,0.0000,0.0000
P00410=0.001,4.491,-0.583,0.0000,0.0000,0.0000
///RCONF 1,0,0,0,1,0,0,0,0,0,0,0,0,0,0,0,0,0,0,0,0,0,0,0
P00411=-0.015,3.627,0.872,0.0000,0.0000,0.0000
P00412=0.002,3.829,0.787,0.0000,0.0000,0.0000
P00413=0.046,0.107,-0.040,0.0000,0.0000,0.0000
///RCONF 1,0,0,0,0,0,0,0,0,0,0,0,0,0,0,0,0,0,0,0,0,0,0,0
P00414=0.046,0.800,0.739,0.0000,0.0000,0.0000
///RCONF 0,0,0,0,0,0,0,0,0,0,0,0,0,0,0,0,0,0,0,0,0,0,0,0
P00415=-1.781,-1.303,3.250,0.0000,0.0000,0.0000
P00416=0.027,1.119,3.078,0.0000,0.0000,0.0000
///RCONF 1,0,0,0,1,0,0,0,0,0,0,0,0,0,0,0,0,0,0,0,0,0,0,0
P00417=0.059,4.721,3.973,0.0000,0.0000,0.0000
//INST
///DATE 2024/05/15 11:40
///ATTR SC,RW
///GROUP1 RB1,BS1
NOP
CALL JOB:MOVE_INTO_TUNNEL
MOVJ C00000 BC00000 VJ=50.00
MOVJ C00001 BC00001 VJ=30.00
MOVJ C00002 BC00002 VJ=30.00
MOVL C00003 BC00003 V=333.3
MOVJ C00004 BC00004 VJ=30.00
MOVL C00005 BC00005 V=500.0
'------------------------
'W31.2
'------------------------
MOVL C00006 BC00006 V=166.7 PL=0
REFP 3 C00007 BC00007
CALL JOB:SEARCH-R1
SET P0300 P0006
SFTON P0300
MOVL C00008 BC00008 V=66.7 PL=0
REFP 3 C00009 BC00009
CALL JOB:SEARCH-R1
SET P0300 P0006
SFTON P0300
MOVL C00010 BC00010 V=166.7 PL=0
SFTOF
'------------------------
'W31.4
'------------------------
MOVL C00011 BC00011 V=666.7
MOVL C00012 BC00012 V=83.3 PL=0
REFP 3 C00013 BC00013
CALL JOB:SEARCH-R1
SET P0301 P0006
SFTON P0301
MOVL C00014 BC00014 V=166.7 PL=0
REFP 3 C00015 BC00015
CALL JOB:SEARCH-R1
SET P0301 P0006
SFTON P0301
MOVL C00016 BC00016 V=166.7 PL=0
SFTOF
'------------------------
'W31.6
'------------------------
MOVL C00017 BC00017 V=666.7
MOVL C00018 BC00018 V=83.3 PL=0
REFP 3 C00019 BC00019
CALL JOB:SEARCH-R1
SET P0302 P0006
SFTON P0302
MOVL C00020 BC00020 V=166.7 PL=0
REFP 3 C00021 BC00021
CALL JOB:SEARCH-R1
SET P0302 P0006
SFTON P0302
MOVL C00022 BC00022 V=250.0 PL=0
SFTOF
'------------------------
'W31.8
'------------------------
MOVL C00023 BC00023 V=666.7
MOVL C00024 BC00024 V=83.3 PL=0
REFP 3 C00025 BC00025
CALL JOB:SEARCH-R1
SET P0303 P0006
SFTON P0303
MOVL C00026 BC00026 V=166.7 PL=0
REFP 3 C00027 BC00027
CALL JOB:SEARCH-R1
SET P0303 P0006
SFTON P0303
MOVL C00028 BC00028 V=250.0 PL=0
SFTOF
'------------------------
'W31.9
'------------------------
MOVL C00029 BC00029 V=666.7
MOVL C00030 BC00030 V=83.3 PL=0
REFP 3 C00031 BC00031
CALL JOB:SEARCH-R1
SET P0304 P0006
SFTON P0304
MOVL C00032 BC00032 V=166.7 PL=0
REFP 3 C00033 BC00033
CALL JOB:SEARCH-R1
SET P0304 P0006
SFTON P0304
MOVL C00034 BC00034 V=250.0 PL=0
SFTOF
'------------------------
'W31.11
'------------------------
MOVL C00035 BC00035 V=666.7
MOVL C00036 BC00036 V=83.3 PL=0
REFP 3 C00037 BC00037
CALL JOB:SEARCH-R1
SET P0305 P0006
SFTON P0305
MOVL C00038 BC00038 V=166.7 PL=0
REFP 3 C00039 BC00039
CALL JOB:SEARCH-R1
SET P0305 P0006
SFTON P0305
MOVL C00040 BC00040 V=250.0 PL=0
SFTOF
'------------------------
'W31.13
'------------------------
MOVL C00041 BC00041 V=666.7
MOVL C00042 BC00042 V=100.0 PL=0
REFP 3 C00043 BC00043
CALL JOB:SEARCH-R1
SET P0306 P0006
SFTON P0306
MOVL C00044 BC00044 V=166.7 PL=0
REFP 3 C00045 BC00045
CALL JOB:SEARCH-R1
SET P0306 P0006
SFTON P0306
MOVL C00046 BC00046 V=250.0 PL=0
SFTOF
'------------------------
'W31.14
'------------------------
MOVL C00047 BC00047 V=666.7
MOVL C00048 BC00048 V=100.0 PL=0
REFP 3 C00049 BC00049
CALL JOB:SEARCH-R1
SET P0307 P0006
SFTON P0307
MOVL C00050 BC00050 V=166.7 PL=0
REFP 3 C00051 BC00051
CALL JOB:SEARCH-R1
SET P0307 P0006
SFTON P0307
MOVL C00052 BC00052 V=250.0 PL=0
SFTOF
'------------------------
'W31.16
'------------------------
MOVL C00053 BC00053 V=666.7
MOVL C00054 BC00054 V=100.0 PL=0
REFP 3 C00055 BC00055
CALL JOB:SEARCH-R1
SET P0308 P0006
SFTON P0308
MOVL C00056 BC00056 V=166.7 PL=0
REFP 3 C00057 BC00057
CALL JOB:SEARCH-R1
SET P0308 P0006
SFTON P0308
MOVL C00058 BC00058 V=250.0 PL=0
SFTOF
MOVL C00059 BC00059 V=166.7
MOVL C00060 BC00060 V=333.3
MOVL C00061 BC00061 V=666.7
MOVL C00062 BC00062 V=500.0
MOVJ C00063 BC00063 VJ=60.00
MOVL C00064 BC00064 V=500.0 PL=0
MOVL C00065 BC00065 V=500.0 PL=0
MOVL C00066 BC00066 V=500.0 PL=0
'------------------------
'W31.18
'------------------------
MOVL C00067 BC00067 V=333.3 PL=0
MOVL C00068 BC00068 V=133.3 PL=0
REFP 3 C00069 BC00069
CALL JOB:SEARCH-R1
SET P0309 P0006
SFTON P0309
MOVL C00070 BC00070 V=166.7 PL=0
REFP 3 C00071 BC00071
CALL JOB:SEARCH-R1
SET P0309 P0006
SFTON P0309
MOVL C00072 BC00072 V=250.0 PL=0
SFTOF
'------------------------
'W31.19
'------------------------
MOVL C00073 BC00073 V=666.7
MOVL C00074 BC00074 V=100.0 PL=0
REFP 3 C00075 BC00075
CALL JOB:SEARCH-R1
SET P0310 P0006
SFTON P0310
MOVL C00076 BC00076 V=166.7 PL=0
REFP 3 C00077 BC00077
CALL JOB:SEARCH-R1
SET P0310 P0006
SFTON P0310
MOVL C00078 BC00078 V=250.0 PL=0
SFTOF
'------------------------
'W31.21
'------------------------
MOVL C00079 BC00079 V=666.7
MOVL C00080 BC00080 V=100.0 PL=0
REFP 3 C00081 BC00081
CALL JOB:SEARCH-R1
SET P0311 P0006
SFTON P0311
MOVL C00082 BC00082 V=166.7 PL=0
REFP 3 C00083 BC00083
CALL JOB:SEARCH-R1
SET P0311 P0006
SFTON P0311
MOVL C00084 BC00084 V=250.0 PL=0
SFTOF
'------------------------
'W31.22
'------------------------
MOVL C00085 BC00085 V=666.7
MOVL C00086 BC00086 V=100.0 PL=0
REFP 3 C00087 BC00087
CALL JOB:SEARCH-R1
SET P0312 P0006
SFTON P0312
MOVL C00088 BC00088 V=166.7 PL=0
REFP 3 C00089 BC00089
CALL JOB:SEARCH-R1
SET P0312 P0006
SFTON P0312
MOVL C00090 BC00090 V=250.0 PL=0
SFTOF
'------------------------
'W31.24
'------------------------
MOVL C00091 BC00091 V=666.7
MOVL C00092 BC00092 V=100.0 PL=0
REFP 3 C00093 BC00093
CALL JOB:SEARCH-R1
SET P0313 P0006
SFTON P0313
MOVL C00094 BC00094 V=166.7 PL=0
REFP 3 C00095 BC00095
CALL JOB:SEARCH-R1
SET P0313 P0006
SFTON P0313
MOVL C00096 BC00096 V=166.7 PL=0
SFTOF
'------------------------
'W31.26
'------------------------
MOVL C00097 BC00097 V=666.7
MOVL C00098 BC00098 V=100.0 PL=0
REFP 3 C00099 BC00099
CALL JOB:SEARCH-R1
SET P0314 P0006
SFTON P0314
MOVL C00100 BC00100 V=166.7 PL=0
REFP 3 C00101 BC00101
CALL JOB:SEARCH-R1
SET P0314 P0006
SFTON P0314
MOVL C00102 BC00102 V=250.0 PL=0
SFTOF
'------------------------
'W31.27
'------------------------
MOVL C00103 BC00103 V=666.7
MOVL C00104 BC00104 V=100.0 PL=0
REFP 3 C00105 BC00105
CALL JOB:SEARCH-R1
SET P0315 P0006
SFTON P0315
MOVL C00106 BC00106 V=166.7 PL=0
REFP 3 C00107 BC00107
CALL JOB:SEARCH-R1
SET P0315 P0006
SFTON P0315
MOVL C00108 BC00108 V=250.0 PL=0
SFTOF
MOVL C00109 BC00109 V=666.7
MOVL C00110 BC00110 V=666.7
MOVL C00111 BC00111 V=666.7
MOVL C00112 BC00112 V=666.7
MOVL C00113 BC00113 V=666.7
MOVL C00114 BC00114 V=666.7
MOVL C00115 BC00115 V=666.7
MOVL C00116 BC00116 V=583.3
MOVL C00117 BC00117 V=500.0
MOVL C00118 BC00118 V=333.3 PL=0
'------------------------
'W31.29
'------------------------
MOVL C00119 BC00119 V=166.7
MOVL C00120 BC00120 V=100.0 PL=0
REFP 3 C00121 BC00121
CALL JOB:SEARCH-R1
SET P0316 P0006
SFTON P0316
MOVL C00122 BC00122 V=166.7 PL=0
REFP 3 C00123 BC00123
CALL JOB:SEARCH-R1
SET P0316 P0006
SFTON P0316
MOVL C00124 BC00124 V=250.0 PL=0
SFTOF
'------------------------
'W31.31
'------------------------
MOVL C00125 BC00125 V=666.7
MOVL C00126 BC00126 V=100.0 PL=0
REFP 3 C00127 BC00127
CALL JOB:SEARCH-R1
SET P0317 P0006
SFTON P0317
MOVL C00128 BC00128 V=166.7 PL=0
REFP 3 C00129 BC00129
CALL JOB:SEARCH-R1
SET P0317 P0006
SFTON P0317
MOVL C00130 BC00130 V=250.0 PL=0
SFTOF
'------------------------
'W31.32
'------------------------
MOVL C00131 BC00131 V=500.0
MOVL C00132 BC00132 V=500.0
MOVL C00133 BC00133 V=500.0
MOVL C00134 BC00134 V=666.7
MOVJ C00135 BC00135 VJ=80.00
MOVJ C00136 BC00136 VJ=80.00
MOVJ C00137 BC00137 VJ=10.00
MOVJ C00138 BC00138 VJ=50.00
MOVJ C00139 BC00139 VJ=50.00
MOVJ C00140 BC00140 VJ=40.00
MOVL C00141 BC00141 V=500.0
SFTOF
'------------------------
'W214A P
'------------------------
MOVL C00142 BC00142 V=100.0 PL=0
REFP 3 C00143 BC00143
CALL JOB:SEARCH-R1
IMOV P0058 V=11.7
SET P0350 P0006
SFTON P0350
REFP 3 C00144 BC00144
CALL JOB:SEARCH-R1
SET P0350 P0006
SFTON P0350
MOVL C00145 BC00145 V=250.0 PL=0
SFTOF
'------------------------
'W214A L
'------------------------
MOVJ C00146 BC00146 VJ=30.00
MOVL C00147 BC00147 V=100.0 PL=0
REFP 3 C00148 BC00148
CALL JOB:SEARCH-R1
IMOV P0058 V=11.7
SET P0351 P0006
SFTON P0351
REFP 3 C00149 BC00149
CALL JOB:SEARCH-R1
SET P0351 P0006
SFTON P0351
MOVL C00150 BC00150 V=250.0 PL=0
SFTOF
'------------------------
'W219A P
'------------------------
MOVJ C00151 BC00151 VJ=40.00
MOVL C00152 BC00152 V=100.0 PL=0
REFP 3 C00153 BC00153
CALL JOB:SEARCH-R1
IMOV P0058 V=11.7
SET P0352 P0006
SFTON P0352
REFP 3 C00154 BC00154
CALL JOB:SEARCH-R1
SET P0352 P0006
SFTON P0352
MOVL C00155 BC00155 V=250.0 PL=0
SFTOF
'------------------------
'W219A L
'------------------------
MOVJ C00156 BC00156 VJ=30.00
MOVL C00157 BC00157 V=66.7 PL=0
REFP 3 C00158 BC00158
CALL JOB:SEARCH-R1
IMOV P0058 V=11.7
SET P0353 P0006
SFTON P0353
REFP 3 C00159 BC00159
CALL JOB:SEARCH-R1
SET P0353 P0006
SFTON P0353
MOVL C00160 BC00160 V=250.0 PL=0
SFTOF
'------------------------
'W213A P
'------------------------
MOVJ C00161 BC00161 VJ=40.00
MOVL C00162 BC00162 V=100.0 PL=0
REFP 3 C00163 BC00163
CALL JOB:SEARCH-R1
IMOV P0058 V=11.7
SET P0354 P0006
SFTON P0354
REFP 3 C00164 BC00164
CALL JOB:SEARCH-R1
SET P0354 P0006
SFTON P0354
MOVL C00165 BC00165 V=250.0 PL=0
SFTOF
'------------------------
'W213A L
'------------------------
MOVJ C00166 BC00166 VJ=40.00
MOVL C00167 BC00167 V=100.0 PL=0
REFP 3 C00168 BC00168
CALL JOB:SEARCH-R1
IMOV P0058 V=11.7
SET P0355 P0006
SFTON P0355
REFP 3 C00169 BC00169
CALL JOB:SEARCH-R1
SET P0355 P0006
SFTON P0355
MOVL C00170 BC00170 V=250.0 PL=0
SFTOF
'------------------------
'W218A P
'------------------------
MOVJ C00171 BC00171 VJ=40.00
MOVL C00172 BC00172 V=100.0 PL=0
REFP 3 C00173 BC00173
CALL JOB:SEARCH-R1
IMOV P0058 V=11.7
SET P0356 P0006
SFTON P0356
REFP 3 C00174 BC00174
CALL JOB:SEARCH-R1
SET P0356 P0006
SFTON P0356
MOVL C00175 BC00175 V=250.0 PL=0
SFTOF
'------------------------
'W218A L
'------------------------
MOVJ C00176 BC00176 VJ=40.00
MOVL C00177 BC00177 V=100.0 PL=0
REFP 3 C00178 BC00178
CALL JOB:SEARCH-R1
IMOV P0058 V=11.7
SET P0357 P0006
SFTON P0357
REFP 3 C00179 BC00179
CALL JOB:SEARCH-R1
SET P0357 P0006
SFTON P0357
MOVL C00180 BC00180 V=250.0 PL=0
SFTOF
'------------------------
'W215A P
'------------------------
MOVJ C00181 BC00181 VJ=40.00
MOVL C00182 BC00182 V=100.0 PL=0
REFP 3 C00183 BC00183
CALL JOB:SEARCH-R1
IMOV P0058 V=11.7
SET P0358 P0006
SFTON P0358
REFP 3 C00184 BC00184
CALL JOB:SEARCH-R1
SET P0358 P0006
SFTON P0358
MOVL C00185 BC00185 V=250.0 PL=0
SFTOF
'------------------------
'W215A L
'------------------------
MOVL C00186 BC00186 V=666.7
MOVL C00187 BC00187 V=100.0 PL=0
REFP 3 C00188 BC00188
CALL JOB:SEARCH-R1
IMOV P0058 V=11.7
SET P0359 P0006
SFTON P0359
REFP 3 C00189 BC00189
CALL JOB:SEARCH-R1
SET P0359 P0006
SFTON P0359
MOVL C00190 BC00190 V=66.7 PL=0
SFTOF
'------------------------
'W217A P
'------------------------
MOVL C00191 BC00191 V=666.7
MOVL C00192 BC00192 V=100.0 PL=0
REFP 3 C00193 BC00193
CALL JOB:SEARCH-R1
IMOV P0058 V=11.7
SET P0360 P0006
SFTON P0360
REFP 3 C00194 BC00194
CALL JOB:SEARCH-R1
SET P0360 P0006
SFTON P0360
MOVL C00195 BC00195 V=250.0 PL=0
SFTOF
'------------------------
'W217A L
'------------------------
MOVL C00196 BC00196 V=666.7
MOVL C00197 BC00197 V=100.0 PL=0
REFP 3 C00198 BC00198
CALL JOB:SEARCH-R1
IMOV P0058 V=11.7
SET P0361 P0006
SFTON P0361
REFP 3 C00199 BC00199
CALL JOB:SEARCH-R1
SET P0361 P0006
SFTON P0361
MOVL C00200 BC00200 V=250.0 PL=0
SFTOF
MOVL C00201 BC00201 V=666.7
MOVL C00202 BC00202 V=833.3
MOVL C00203 BC00203 V=833.3
MOVJ C00204 BC00204 VJ=70.00
MOVJ C00205 BC00205 VJ=80.00
MOVJ C00206 BC00206 VJ=50.00
MOVJ C00207 BC00207 VJ=50.00
MOVJ C00208 BC00208 VJ=30.00
MOVJ C00209 BC00209 VJ=30.00
'KKK
MOVL C00210 BC00210 V=666.7
MOVL C00211 BC00211 V=666.7
MOVL C00212 BC00212 V=500.0
'------------------------
'W27.4
'------------------------
MOVL C00213 BC00213 V=100.0 PL=0
REFP 3 C00214 BC00214
CALL JOB:SEARCH-R1
SET P0401 P0006
SFTON P0401
MOVL C00215 BC00215 V=166.7 PL=0
REFP 3 C00216 BC00216
CALL JOB:SEARCH-R1
SET P0401 P0006
SFTON P0401
MOVL C00217 BC00217 V=250.0 PL=0
SFTOF
'------------------------
'W27.6
'------------------------
MOVL C00218 BC00218 V=666.7
MOVL C00219 BC00219 V=100.0 PL=0
REFP 3 C00220 BC00220
CALL JOB:SEARCH-R1
SET P0402 P0006
SFTON P0402
MOVL C00221 BC00221 V=100.0 PL=0
REFP 3 C00222 BC00222
CALL JOB:SEARCH-R1
SET P0402 P0006
SFTON P0402
MOVL C00223 BC00223 V=250.0 PL=0
SFTOF
MOVL C00224 BC00224 V=666.7
MOVL C00225 BC00225 V=666.7
'------------------------
'W27.8
'------------------------
MOVL C00226 BC00226 V=666.7
MOVL C00227 BC00227 V=166.7 PL=0
REFP 3 C00228 BC00228
CALL JOB:SEARCH-R1
SET P0403 P0006
SFTON P0403
MOVL C00229 BC00229 V=166.7 PL=0
REFP 3 C00230 BC00230
CALL JOB:SEARCH-R1
SET P0403 P0006
SFTON P0403
MOVL C00231 BC00231 V=250.0 PL=0
SFTOF
'ZMIENNA
GETE D040 P0403 (1)
GETE D041 P0403 (2)
GETE D042 P0403 (3)
SETE P0404 (1) D040
SETE P0404 (2) D041
SETE P0404 (3) D042
COMM '------------------------
COMM 'W27.9
COMM '------------------------
COMM MOVL C00232 BC00232 V=333.3
COMM MOVL C00233 BC00233 V=66.7 PL=0
COMM REFP 3 C00234 BC00234
COMM CALL JOB:SEARCH-R1
COMM SET P0404 P0006
COMM SFTON P0404
COMM MOVL C00235 BC00235 V=66.7 PL=0
COMM REFP 3 C00236 BC00236
COMM CALL JOB:SEARCH-R1
COMM SET P0404 P0006
COMM SFTON P0404
COMM MOVL C00237 BC00237 V=66.7 PL=0
COMM SFTOF
MOVL C00238 BC00238 V=666.7
MOVL C00239 BC00239 V=666.7
MOVJ C00240 BC00240 VJ=30.00
'------------------------
'W27.11
'------------------------
MOVL C00241 BC00241 V=500.0
MOVL C00242 BC00242 V=100.0 PL=0
REFP 3 C00243 BC00243
CALL JOB:SEARCH-R1
SET P0405 P0006
SFTON P0405
MOVL C00244 BC00244 V=166.7 PL=0
REFP 3 C00245 BC00245
CALL JOB:SEARCH-R1
SET P0405 P0006
SFTON P0405
MOVL C00246 BC00246 V=250.0 PL=0
SFTOF
MOVL C00247 BC00247 V=666.7
'------------------------
'W27.13
'------------------------
MOVL C00248 BC00248 V=666.7
MOVL C00249 BC00249 V=666.7
MOVL C00250 BC00250 V=166.7 PL=0
REFP 3 C00251 BC00251
CALL JOB:SEARCH-R1
SET P0406 P0006
SFTON P0406
MOVL C00252 BC00252 V=166.7 PL=0
REFP 3 C00253 BC00253
CALL JOB:SEARCH-R1
SET P0406 P0006
SFTON P0406
MOVL C00254 BC00254 V=250.0 PL=0
SFTOF
'------------------------
'W27.14
'------------------------
MOVL C00255 BC00255 V=666.7
MOVL C00256 BC00256 V=100.0 PL=0
REFP 3 C00257 BC00257
CALL JOB:SEARCH-R1
SET P0407 P0006
SFTON P0407
MOVL C00258 BC00258 V=166.7 PL=0
REFP 3 C00259 BC00259
CALL JOB:SEARCH-R1
SET P0407 P0006
SFTON P0407
MOVL C00260 BC00260 V=250.0 PL=0
SFTOF
'------------------------
'W27.16
'------------------------
MOVL C00261 BC00261 V=666.7
MOVL C00262 BC00262 V=100.0 PL=0
REFP 3 C00263 BC00263
CALL JOB:SEARCH-R1
SET P0408 P0006
SFTON P0408
MOVL C00264 BC00264 V=166.7 PL=0
REFP 3 C00265 BC00265
CALL JOB:SEARCH-R1
SET P0408 P0006
SFTON P0408
MOVL C00266 BC00266 V=250.0 PL=0
MOVL C00267 BC00267 V=666.7
SFTOF
'------------------------
'W27.18
'------------------------
MOVJ C00268 BC00268 VJ=40.00
MOVJ C00269 BC00269 VJ=50.00
MOVL C00270 BC00270 V=666.7
MOVL C00271 BC00271 V=333.3
MOVL C00272 BC00272 V=100.0 PL=0
REFP 3 C00273 BC00273
CALL JOB:SEARCH-R1
SET P0409 P0006
SFTON P0409
MOVL C00274 BC00274 V=16.7 PL=0
REFP 3 C00275 BC00275
CALL JOB:SEARCH-R1
SET P0409 P0006
SFTON P0409
MOVL C00276 BC00276 V=166.7 PL=0
SFTOF
'------------------------
'W27.19
'------------------------
MOVL C00277 BC00277 V=666.7
MOVL C00278 BC00278 V=100.0 PL=0
REFP 3 C00279 BC00279
CALL JOB:SEARCH-R1
SET P0410 P0006
SFTON P0410
MOVL C00280 BC00280 V=166.7 PL=0
REFP 3 C00281 BC00281
CALL JOB:SEARCH-R1
SET P0410 P0006
SFTON P0410
MOVL C00282 BC00282 V=250.0 PL=0
SFTOF
'------------------------
'W27.21
'------------------------
MOVL C00283 BC00283 V=666.7
MOVL C00284 BC00284 V=100.0 PL=0
REFP 3 C00285 BC00285
CALL JOB:SEARCH-R1
SET P0411 P0006
SFTON P0411
MOVL C00286 BC00286 V=166.7 PL=0
REFP 3 C00287 BC00287
CALL JOB:SEARCH-R1
SET P0411 P0006
SFTON P0411
MOVL C00288 BC00288 V=166.7 PL=0
SFTOF
'------------------------
'W27.22
'------------------------
MOVL C00289 BC00289 V=666.7
MOVL C00290 BC00290 V=100.0 PL=0
REFP 3 C00291 BC00291
CALL JOB:SEARCH-R1
SET P0412 P0006
SFTON P0412
MOVL C00292 BC00292 V=166.7 PL=0
REFP 3 C00293 BC00293
CALL JOB:SEARCH-R1
SET P0412 P0006
SFTON P0412
MOVL C00294 BC00294 V=166.7 PL=0
SFTOF
'------------------------
'W27.24
'------------------------
MOVL C00295 BC00295 V=666.7
MOVL C00296 BC00296 V=100.0 PL=0
REFP 3 C00297 BC00297
CALL JOB:SEARCH-R1
SET P0413 P0006
SFTON P0413
MOVL C00298 BC00298 V=166.7 PL=0
REFP 3 C00299 BC00299
CALL JOB:SEARCH-R1
SET P0413 P0006
SFTON P0413
MOVL C00300 BC00300 V=250.0 PL=0
SFTOF
GETE D040 P0413 (1)
GETE D041 P0413 (2)
GETE D042 P0413 (3)
SETE P0414 (1) D040
SETE P0414 (2) D041
SETE P0414 (3) D042
GETE D040 P0413 (1)
GETE D041 P0413 (2)
GETE D042 P0413 (3)
SETE P0415 (1) D040
SETE P0415 (2) D041
SETE P0415 (3) D042
COMM '------------------------
COMM 'W27.26
COMM '------------------------
COMM MOVL C00301 BC00301 V=333.3
COMM MOVL C00302 BC00302 V=66.7 PL=0
COMM REFP 3 C00303 BC00303
COMM CALL JOB:SEARCH-R1
COMM SET P0414 P0006
COMM SFTON P0414
COMM MOVL C00304 BC00304 V=66.7 PL=0
COMM REFP 3 C00305 BC00305
COMM CALL JOB:SEARCH-R1
COMM SET P0414 P0006
COMM SFTON P0414
COMM MOVL C00306 BC00306 V=66.7 PL=0
COMM SFTOF
MOVL C00307 BC00307 V=333.3
MOVL C00308 BC00308 V=666.7
MOVL C00309 BC00309 V=1000.0
MOVL C00310 BC00310 V=1000.0
MOVL C00311 BC00311 V=666.7
MOVL C00312 BC00312 V=500.0
'------------------------
'W27.29
'------------------------
MOVL C00313 BC00313 V=333.3
MOVL C00314 BC00314 V=100.0 PL=0
REFP 3 C00315 BC00315
CALL JOB:SEARCH-R1
SET P0416 P0006
SFTON P0416
MOVL C00316 BC00316 V=166.7 PL=0
REFP 3 C00317 BC00317
CALL JOB:SEARCH-R1
SET P0416 P0006
SFTON P0416
MOVL C00318 BC00318 V=250.0 PL=0
SFTOF
'------------------------
'W27.31
'------------------------
MOVL C00319 BC00319 V=666.7
MOVL C00320 BC00320 V=100.0 PL=0
REFP 3 C00321 BC00321
CALL JOB:SEARCH-R1
SET P0417 P0006
SFTON P0417
MOVL C00322 BC00322 V=166.7 PL=0
REFP 3 C00323 BC00323
CALL JOB:SEARCH-R1
SET P0417 P0006
SFTON P0417
MOVL C00324 BC00324 V=250.0 PL=0
SFTOF
'------------------------
'W27.32
'------------------------
SFTOF
MOVL C00325 BC00325 V=666.7
MOVJ C00326 BC00326 VJ=80.00
CALL JOB:FRONT_SEARCH_90ST-1_5040
MOVJ C00327 BC00327 VJ=50.00
MOVJ C00328 BC00328 VJ=40.00
MOVJ C00329 BC00329 VJ=40.00
MOVL C00330 BC00330 V=500.0
MOVJ C00331 BC00331 VJ=30.00
'------------------------
'W31.2
'------------------------
SFTON P0300
MOVL C00332 BC00332 V=500.0
MOVL C00333 BC00333 V=133.3 PL=0
MACRO1 MJ#(0) ARGF10
ARCON
MOVL C00334 BC00334 V=10.8
ARCOF
MOVL C00335 BC00335 V=250.0
SFTOF
'------------------------
'W31.4
'------------------------
SFTON P0301
MOVL C00336 BC00336 V=500.0
MOVL C00337 BC00337 V=166.7
MACRO1 MJ#(0) ARGF10
ARCON
MOVL C00338 BC00338 V=10.8
ARCOF
MOVL C00339 BC00339 V=250.0
SFTOF
'------------------------
'W31.6
'------------------------
SFTON P0302
MOVL C00340 BC00340 V=500.0
MOVL C00341 BC00341 V=166.7 PL=0
MACRO1 MJ#(0) ARGF10
ARCON
MOVL C00342 BC00342 V=10.8
ARCOF
MOVL C00343 BC00343 V=166.7
SFTOF
'------------------------
'W31.8
'------------------------
SFTON P0303
MOVL C00344 BC00344 V=500.0
MOVL C00345 BC00345 V=166.7 PL=0
MACRO1 MJ#(0) ARGF10
ARCON
MOVL C00346 BC00346 V=10.8
ARCOF
MOVL C00347 BC00347 V=166.7
SFTOF
'------------------------
'W31.9
'------------------------
SFTON P0304
MOVL C00348 BC00348 V=500.0
MOVL C00349 BC00349 V=166.7 PL=0
MACRO1 MJ#(0) ARGF10
ARCON
MOVL C00350 BC00350 V=10.8
ARCOF
MOVL C00351 BC00351 V=166.7
SFTOF
MOVL C00352 BC00352 V=500.0
MOVL C00353 BC00353 V=666.7
MOVJ C00354 BC00354 VJ=30.00
MOVJ C00355 BC00355 VJ=50.00
'::::::::::::::::::::::::::::::::
'::::::::::::::::::::::::::::::::
'::::::::::::::::::::::::::::::::
'::::::::::::::::::::::::::::::::
'::::::::::::::::::::::::::::::::
MOVJ C00356 BC00356 VJ=30.00
MOVJ C00357 BC00357 VJ=30.00
MOVJ C00358 BC00358 VJ=25.00
MOVJ C00359 BC00359 VJ=30.00
MOVJ C00360 BC00360 VJ=40.00
MOVJ C00361 BC00361 VJ=40.00
'------------------------
'W27.1
'------------------------
MOVL C00362 BC00362 V=666.7
MOVL C00363 BC00363 V=166.7 PL=0
MACRO1 MJ#(0) ARGF9
ARCOF
SFTOF
'BELKA PRZEJAZD
MOVL C00364 BC00364 V=333.3
MOVJ C00365 BC00365 VJ=30.00
MOVJ C00366 BC00366 VJ=30.00
MOVJ C00367 BC00367 VJ=40.00
MOVJ C00368 BC00368 VJ=50.00
MOVJ C00369 BC00369 VJ=50.00
MOVJ C00370 BC00370 VJ=50.00
MOVL C00371 BC00371 V=166.7
'------------------------
'W213A
'------------------------
SFTON P0355
MOVL C00372 BC00372 V=500.0
MOVL C00373 BC00373 V=166.7 PL=0
MACRO1 MJ#(0) ARGF14
ARCON
SFTOF
SFTON P0354
MOVL C00374 BC00374 V=11.7
ARCOF
MOVL C00375 BC00375 V=166.7
SFTOF
MOVJ C00376 BC00376 VJ=50.00
MOVJ C00377 BC00377 VJ=80.00
MOVJ C00378 BC00378 VJ=10.00
MOVJ C00379 BC00379 VJ=40.00
MOVJ C00380 BC00380 VJ=40.00
MOVJ C00381 BC00381 VJ=30.00
MOVJ C00382 BC00382 VJ=30.00
'5.5.1
'------------------------
'W31.11
'------------------------
SFTON P0305
MOVL C00383 BC00383 V=333.3
MOVL C00384 BC00384 V=166.7
MACRO1 MJ#(0) ARGF10
ARCON
MOVL C00385 BC00385 V=10.8
ARCOF
MOVL C00386 BC00386 V=166.7
SFTOF
'------------------------
'W31.13
'------------------------
SFTON P0306
MOVL C00387 BC00387 V=333.3
MOVL C00388 BC00388 V=166.7
ARCON
MOVL C00389 BC00389 V=10.8
ARCOF
MOVL C00390 BC00390 V=166.7
SFTOF
'------------------------
'W31.14
'------------------------
SFTON P0307
MOVL C00391 BC00391 V=333.3
MOVL C00392 BC00392 V=166.7 PL=0
ARCON
MOVL C00393 BC00393 V=10.8
ARCOF
MOVL C00394 BC00394 V=250.0
SFTOF
MOVL C00395 BC00395 V=500.0
MOVL C00396 BC00396 V=500.0
MOVJ C00397 BC00397 VJ=30.00
MOVJ C00398 BC00398 VJ=30.00
MOVJ C00399 BC00399 VJ=30.00
MOVJ C00400 BC00400 VJ=40.00
'::::::::::::::::::::::::::::::::
'::::::::::::::::::::::::::::::::
'------------------------
'W27.9
'------------------------
'::::::::::::::::::::::::::::::::
'::::::::::::::::::::::::::::::::
MOVJ C00401 BC00401 VJ=40.00
MOVJ C00402 BC00402 VJ=30.00
MOVL C00403 BC00403 V=666.7
SFTON P0404
MOVL C00404 BC00404 V=500.0
MOVL C00405 BC00405 V=200.0 PL=0
MACRO1 MJ#(0) ARGF24
ARCON
MOVL C00406 BC00406 V=7.5
ARCOF
MOVL C00407 BC00407 V=166.7
SFTOF
MOVL C00408 BC00408 V=500.0
MOVL C00409 BC00409 V=500.0
MOVJ C00410 BC00410 VJ=50.00
'------------------------
'W27.11
'------------------------
MOVL C00411 BC00411 V=500.0
SFTON P0405
MOVL C00412 BC00412 V=333.3
MOVL C00413 BC00413 V=200.0 PL=0
MACRO1 MJ#(0) ARGF24
ARCON
MOVL C00414 BC00414 V=7.5
ARCOF
MOVL C00415 BC00415 V=166.7
SFTOF
MOVL C00416 BC00416 V=166.7
'------------------------
'W27.13
'------------------------
SFTON P0406
MOVL C00417 BC00417 V=333.3
MOVL C00418 BC00418 V=133.3 PL=0
MACRO1 MJ#(0) ARGF24
ARCON
MOVL C00419 BC00419 V=7.5
ARCOF
MOVL C00420 BC00420 V=250.0
SFTOF
MOVJ C00421 BC00421 VJ=30.00
MOVJ C00422 BC00422 VJ=50.00
MOVJ C00423 BC00423 VJ=50.00
'::::::::::::::::::::::::
'::::::::::::::::::::::::
'::::::::::::::::::::::::
'::::::::::::::::::::::::
'::::::::::::::::::::::::
'::::::::::::::::::::::::
'::::::::::::::::::::::::
MOVJ C00424 BC00424 VJ=50.00
MOVJ C00425 BC00425 VJ=30.00
'------------------------
'W214A
'------------------------
SFTON P0351
MOVL C00426 BC00426 V=333.3
MOVL C00427 BC00427 V=500.0
MOVL C00428 BC00428 V=166.7 PL=0
MACRO1 MJ#(0) ARGF14
ARCON
SFTOF
SFTON P0350
MOVL C00429 BC00429 V=11.7
ARCOF
MOVL C00430 BC00430 V=250.0
SFTOF
MOVJ C00431 BC00431 VJ=50.00
MOVJ C00432 BC00432 VJ=50.00
MOVJ C00433 BC00433 VJ=10.00
MOVJ C00434 BC00434 VJ=50.00
MOVJ C00435 BC00435 VJ=50.00
MOVJ C00436 BC00436 VJ=50.00
MOVJ C00437 BC00437 VJ=30.00
MOVJ C00438 BC00438 VJ=20.00
'------------------------
'W31.16
MACRO1 MJ#(0) ARGF10
'------------------------
SFTON P0308
MOVL C00439 BC00439 V=333.3
MOVL C00440 BC00440 V=66.7 PL=0
ARCON
MOVL C00441 BC00441 V=10.8
ARCOF
MOVL C00442 BC00442 V=250.0
SFTOF
MOVL C00443 BC00443 V=500.0
MOVL C00444 BC00444 V=500.0
MOVL C00445 BC00445 V=666.7
MOVL C00446 BC00446 V=833.3
MOVL C00447 BC00447 V=666.7
MOVL C00448 BC00448 V=666.7
MOVL C00449 BC00449 V=333.3
MOVL C00450 BC00450 V=333.3
MOVL C00451 BC00451 V=333.3
MOVL C00452 BC00452 V=333.3
'------------------------
'W31.18
'------------------------
SFTON P0309
MOVL C00453 BC00453 V=166.7
MOVL C00454 BC00454 V=166.7 PL=0
ARCON
MOVL C00455 BC00455 V=10.8
ARCOF
MOVL C00456 BC00456 V=166.7
SFTOF
'------------------------
'W31.19
'------------------------
SFTON P0310
MOVL C00457 BC00457 V=333.3
MOVL C00458 BC00458 V=166.7 PL=0
MACRO1 MJ#(0) ARGF10
ARCON
MOVL C00459 BC00459 V=10.8
ARCOF
MOVL C00460 BC00460 V=250.0
SFTOF
MOVL C00461 BC00461 V=250.0
MOVL C00462 BC00462 V=500.0
MOVL C00463 BC00463 V=666.7
MOVL C00464 BC00464 V=666.7
MOVJ C00465 BC00465 VJ=50.00
'::::::::::::::::::::::::
'::::::::::::::::::::::::
'::::::::::::::::::::::::
'::::::::::::::::::::::::
'::::::::::::::::::::::::
'::::::::::::::::::::::::
'::::::::::::::::::::::::
MOVJ C00466 BC00466 VJ=50.00
MOVJ C00467 BC00467 VJ=40.00
'::::::::::::::::::::::::::::::::
'::::::::::::::::::::::::::::::::
'------------------------
'W27.14
'------------------------
'::::::::::::::::::::::::::::::::
'::::::::::::::::::::::::::::::::
SFTON P0407
MOVJ C00468 BC00468 VJ=40.00
MOVL C00469 BC00469 V=500.0
MOVL C00470 BC00470 V=166.7 PL=0
MACRO1 MJ#(0) ARGF24
ARCON
MOVL C00471 BC00471 V=6.7
ARCOF
MOVL C00472 BC00472 V=250.0
SFTOF
'------------------------
'W27.16
'------------------------
SFTON P0408
MOVL C00473 BC00473 V=333.3
MOVL C00474 BC00474 V=166.7 PL=0
MACRO1 MJ#(0) ARGF24
ARCON
MOVL C00475 BC00475 V=6.7
ARCOF
MOVL C00476 BC00476 V=250.0
SFTOF
MOVL C00477 BC00477 V=500.0
MOVL C00478 BC00478 V=500.0
MOVJ C00479 BC00479 VJ=40.00
MOVJ C00480 BC00480 VJ=40.00
MOVL C00481 BC00481 V=666.7
'------------------------
'W27.18
'------------------------
SFTON P0409
MOVL C00482 BC00482 V=500.0
MOVL C00483 BC00483 V=166.7 PL=0
MACRO1 MJ#(0) ARGF24
ARCON
MOVL C00484 BC00484 V=7.5
ARCOF
MOVL C00485 BC00485 V=250.0
SFTOF
MOVJ C00486 BC00486 VJ=20.00
MOVJ C00487 BC00487 VJ=30.00
MOVJ C00488 BC00488 VJ=50.00
'::::::::::::::::::::::::
'::::::::::::::::::::::::
'::::::::::::::::::::::::
'::::::::::::::::::::::::
'::::::::::::::::::::::::
'::::::::::::::::::::::::
'::::::::::::::::::::::::
MOVJ C00489 BC00489 VJ=50.00
MOVJ C00490 BC00490 VJ=50.00
'------------------------
'W215A
'------------------------
SFTON P0359
MOVL C00491 BC00491 V=666.7
MOVL C00492 BC00492 V=166.7 PL=0
MACRO1 MJ#(0) ARGF14
ARCON
SFTOF
SFTON P0358
MOVL C00493 BC00493 V=11.7
ARCOF
MOVL C00494 BC00494 V=333.3
SFTOF
MOVJ C00495 BC00495 VJ=30.00
MOVJ C00496 BC00496 VJ=50.00
MOVJ C00497 BC00497 VJ=50.00
MOVJ C00498 BC00498 VJ=50.00
MOVJ C00499 BC00499 VJ=50.00
MOVJ C00500 BC00500 VJ=50.00
MOVJ C00501 BC00501 VJ=30.00
MOVJ C00502 BC00502 VJ=30.00
'------------------------
'W31.21
'------------------------
SFTON P0311
MOVL C00503 BC00503 V=666.7
MOVL C00504 BC00504 V=166.7 PL=0
MACRO1 MJ#(0) ARGF10
ARCON
MOVL C00505 BC00505 V=10.8
ARCOF
MOVL C00506 BC00506 V=250.0
SFTOF
'------------------------
'W31.22
'------------------------
SFTON P0312
MOVL C00507 BC00507 V=333.3
MOVL C00508 BC00508 V=166.7 PL=0
ARCON
MOVL C00509 BC00509 V=10.8
ARCOF
MOVL C00510 BC00510 V=250.0
SFTOF
'------------------------
'W31.24
'------------------------
SFTON P0313
MOVL C00511 BC00511 V=500.0
MOVL C00512 BC00512 V=166.7 PL=0
MACRO1 MJ#(0) ARGF10
ARCON
MOVL C00513 BC00513 V=10.8
ARCOF
MOVL C00514 BC00514 V=250.0
MOVL C00515 BC00515 V=333.3
MOVL C00516 BC00516 V=500.0
SFTOF
MOVL C00517 BC00517 V=666.7
MOVJ C00518 BC00518 VJ=50.00
MOVJ C00519 BC00519 VJ=50.00
MOVJ C00520 BC00520 VJ=50.00
'::::::::::::::::::::::::
'::::::::::::::::::::::::
'::::::::::::::::::::::::
'::::::::::::::::::::::::
'::::::::::::::::::::::::
'::::::::::::::::::::::::
'::::::::::::::::::::::::
MOVJ C00521 BC00521 VJ=50.00
MOVJ C00522 BC00522 VJ=30.00
MOVJ C00523 BC00523 VJ=30.00
MOVJ C00524 BC00524 VJ=30.00
'::::::::::::::::::::::::::::::::
'::::::::::::::::::::::::::::::::
'------------------------
'W27.19
'------------------------
'::::::::::::::::::::::::::::::::
'::::::::::::::::::::::::::::::::
SFTOF
MOVL C00525 BC00525 V=666.7
MOVL C00526 BC00526 V=666.7
MOVL C00527 BC00527 V=666.7
SFTON P0410
MOVL C00528 BC00528 V=166.7 PL=0
MACRO1 MJ#(0) ARGF24
ARCON
MOVL C00529 BC00529 V=7.5
ARCOF
MOVL C00530 BC00530 V=333.3
SFTOF
MOVJ C00531 BC00531 VJ=30.00
MOVJ C00532 BC00532 VJ=50.00
MOVJ C00533 BC00533 VJ=50.00
MOVJ C00534 BC00534 VJ=50.00
MOVJ C00535 BC00535 VJ=50.00
MOVJ C00536 BC00536 VJ=30.00
'------------------------
'W27.21
'------------------------
SFTON P0411
MOVL C00537 BC00537 V=333.3
MOVL C00538 BC00538 V=166.7 PL=0
MACRO1 MJ#(0) ARGF24
ARCON
MOVL C00539 BC00539 V=7.5
ARCOF
MOVL C00540 BC00540 V=333.3
SFTOF
'------------------------
'W27.22
'------------------------
SFTON P0412
MOVL C00541 BC00541 V=333.3
MOVL C00542 BC00542 V=166.7 PL=0
MACRO1 MJ#(0) ARGF24
ARCON
MOVL C00543 BC00543 V=7.5
ARCOF
SFTOF
MOVL C00544 BC00544 V=250.0
SFTOF
'::::::::::::::::::::::::
'::::::::::::::::::::::::
'::::::::::::::::::::::::
'::::::::::::::::::::::::
'::::::::::::::::::::::::
'::::::::::::::::::::::::
'::::::::::::::::::::::::
MOVJ C00545 BC00545 VJ=30.00
MOVJ C00546 BC00546 VJ=40.00
MOVJ C00547 BC00547 VJ=80.00
MOVJ C00548 BC00548 VJ=80.00
'------------------------
'W215A
'------------------------
MOVJ C00549 BC00549 VJ=80.00
MOVJ C00550 BC00550 VJ=80.00
SFTON P0360
MOVL C00551 BC00551 V=500.0
MOVL C00552 BC00552 V=666.7
MOVL C00553 BC00553 V=166.7 PL=0
MACRO1 MJ#(0) ARGF14
ARCON
SFTOF
SFTON P0361
MOVL C00554 BC00554 V=11.7
ARCOF
MOVL C00555 BC00555 V=333.3
SFTOF
MOVJ C00556 BC00556 VJ=50.00
MOVJ C00557 BC00557 VJ=50.00
MOVJ C00558 BC00558 VJ=50.00
MOVJ C00559 BC00559 VJ=60.00
MOVJ C00560 BC00560 VJ=50.00
MOVJ C00561 BC00561 VJ=50.00
MOVJ C00562 BC00562 VJ=30.00
MOVJ C00563 BC00563 VJ=20.00
MOVJ C00564 BC00564 VJ=20.00
'------------------------
'W31.26
'------------------------
SFTON P0314
MOVL C00565 BC00565 V=666.7
MOVL C00566 BC00566 V=166.7 PL=0
MACRO1 MJ#(0) ARGF10
ARCON
MOVL C00567 BC00567 V=10.8
ARCOF
MOVL C00568 BC00568 V=166.7
SFTOF
'------------------------
'W31.27
'------------------------
SFTON P0315
MOVL C00569 BC00569 V=166.7 PL=0
MACRO1 MJ#(0) ARGF10
ARCON
MOVL C00570 BC00570 V=10.8
ARCOF
MOVL C00571 BC00571 V=250.0
SFTOF
SFTOF
MOVL C00572 BC00572 V=333.3
MOVL C00573 BC00573 V=333.3
MOVL C00574 BC00574 V=333.3
MOVJ C00575 BC00575 VJ=50.00
MOVJ C00576 BC00576 VJ=50.00
MOVJ C00577 BC00577 VJ=40.00
MOVJ C00578 BC00578 VJ=50.00
'::::::::::::::::::::::::
'::::::::::::::::::::::::
'::::::::::::::::::::::::
'::::::::::::::::::::::::
'::::::::::::::::::::::::
'::::::::::::::::::::::::
'::::::::::::::::::::::::
MOVJ C00579 BC00579 VJ=50.00
MOVJ C00580 BC00580 VJ=50.00
'::::::::::::::::::::::::::::::::
'::::::::::::::::::::::::::::::::
'------------------------
'W27.24
'------------------------
'::::::::::::::::::::::::::::::::
'::::::::::::::::::::::::::::::::
SFTON P0413
MOVL C00581 BC00581 V=666.7
MOVL C00582 BC00582 V=166.7 PL=0
MACRO1 MJ#(0) ARGF24
ARCON
MOVL C00583 BC00583 V=7.5
ARCOF
MOVL C00584 BC00584 V=250.0
SFTOF
'------------------------
'W27.26
'------------------------
SFTON P0414
MOVL C00585 BC00585 V=333.3
MOVL C00586 BC00586 V=66.7 PL=0
MACRO1 MJ#(0) ARGF24
ARCON
MOVL C00587 BC00587 V=7.5
ARCOF
MOVL C00588 BC00588 V=250.0
SFTOF
COMM '------------------------
COMM 'W27.27
COMM '------------------------
COMM SFTON P0414
COMM MOVL C00589 BC00589 V=333.3
COMM MOVL C00590 BC00590 V=66.7 PL=0
COMM MACRO1 MJ#(0) ARGF24
COMM ARCON
COMM MOVL C00591 BC00591 V=6.7
COMM ARCOF
COMM MOVL C00592 BC00592 V=83.3
COMM SFTOF
MOVL C00593 BC00593 V=333.3
'::::::::::::::::::::::::
'::::::::::::::::::::::::
'::::::::::::::::::::::::
'::::::::::::::::::::::::
'::::::::::::::::::::::::
'::::::::::::::::::::::::
'::::::::::::::::::::::::
MOVL C00594 BC00594 V=666.7
MOVJ C00595 BC00595 VJ=40.00
MOVJ C00596 BC00596 VJ=40.00
MOVJ C00597 BC00597 VJ=40.00
MOVJ C00598 BC00598 VJ=40.00
'------------------------
'W218A
'------------------------
MOVJ C00599 BC00599 VJ=50.00
MOVJ C00600 BC00600 VJ=50.00
SFTON P0357
MOVL C00601 BC00601 V=666.7
MOVL C00602 BC00602 V=666.7
MOVL C00603 BC00603 V=166.7 PL=0
MACRO1 MJ#(0) ARGF14
ARCON
SFTOF
SFTON P0356
MOVL C00604 BC00604 V=11.7
ARCOF
MOVL C00605 BC00605 V=333.3
MOVL C00606 BC00606 V=500.0
SFTOF
MOVJ C00607 BC00607 VJ=50.00
MOVJ C00608 BC00608 VJ=50.00
MOVJ C00609 BC00609 VJ=50.00
MOVJ C00610 BC00610 VJ=50.00
MOVJ C00611 BC00611 VJ=50.00
MOVJ C00612 BC00612 VJ=30.00
MOVL C00613 BC00613 V=666.7
'------------------------
'W31.29
'------------------------
SFTON P0316
MOVL C00614 BC00614 V=333.3
MOVL C00615 BC00615 V=333.3
MOVL C00616 BC00616 V=333.3
MOVL C00617 BC00617 V=66.7 PL=0
MACRO1 MJ#(0) ARGF10
ARCON
MOVL C00618 BC00618 V=10.8
ARCOF
MOVL C00619 BC00619 V=250.0
SFTOF
'------------------------
'W31.31
'------------------------
SFTON P0317
MOVL C00620 BC00620 V=666.7
MOVL C00621 BC00621 V=166.7 PL=0
ARCON
MOVL C00622 BC00622 V=10.8
ARCOF
MOVL C00623 BC00623 V=250.0
SFTOF
'------------------------
'W31.32
'------------------------
SFTON P0317
MOVL C00624 BC00624 V=333.3 PL=0
MOVL C00625 BC00625 V=166.7 PL=0
ARCON
MOVL C00626 BC00626 V=10.8
ARCOF
MOVL C00627 BC00627 V=250.0
SFTOF
MOVL C00628 BC00628 V=333.3
MOVL C00629 BC00629 V=333.3
MOVL C00630 BC00630 V=500.0
MOVL C00631 BC00631 V=500.0
MOVL C00632 BC00632 V=500.0
MOVJ C00633 BC00633 VJ=40.00
MOVJ C00634 BC00634 VJ=40.00
MOVJ C00635 BC00635 VJ=40.00
MOVJ C00636 BC00636 VJ=40.00
'::::::::::::::::::::::::
'::::::::::::::::::::::::
'::::::::::::::::::::::::
'::::::::::::::::::::::::
'::::::::::::::::::::::::
'::::::::::::::::::::::::
'::::::::::::::::::::::::
MOVJ C00637 BC00637 VJ=40.00
MOVJ C00638 BC00638 VJ=40.00
MOVJ C00639 BC00639 VJ=40.00
'::::::::::::::::::::::::::::::::
'::::::::::::::::::::::::::::::::
'------------------------
'W27.29
'------------------------
'::::::::::::::::::::::::::::::::
'::::::::::::::::::::::::::::::::
SFTON P0416
MOVL C00640 BC00640 V=500.0
MOVL C00641 BC00641 V=66.7 PL=0
MACRO1 MJ#(0) ARGF24
ARCON
MOVL C00642 BC00642 V=7.5
ARCOF
MOVL C00643 BC00643 V=250.0
SFTOF
'------------------------
'W27.31
'------------------------
SFTOF
'::::::::::::::::::::::::
'::::::::::::::::::::::::
'::::::::::::::::::::::::
'::::::::::::::::::::::::
'::::::::::::::::::::::::
'::::::::::::::::::::::::
'::::::::::::::::::::::::
MOVL C00644 BC00644 V=500.0
MOVJ C00645 BC00645 VJ=50.00
MOVJ C00646 BC00646 VJ=50.00
MOVJ C00647 BC00647 VJ=50.00
MOVJ C00648 BC00648 VJ=50.00
MOVJ C00649 BC00649 VJ=50.00
'------------------------
'W219A
'------------------------
MOVJ C00650 BC00650 VJ=50.00
MOVJ C00651 BC00651 VJ=50.00
SFTON P0353
MOVL C00652 BC00652 V=500.0
MOVL C00653 BC00653 V=333.3
MOVL C00654 BC00654 V=166.7 PL=0
MACRO1 MJ#(0) ARGF14
ARCON
SFTOF
SFTON P0352
MOVL C00655 BC00655 V=11.7
ARCOF
MOVL C00656 BC00656 V=250.0
SFTOF
MOVJ C00657 BC00657 VJ=40.00
MOVJ C00658 BC00658 VJ=50.00
CALL JOB:FRONT_WELD_90ST-1_5040
CALL JOB:MOVE_OUT_OF_TUNNEL
END
